LIN {X 0,Y 520.431,Z 549.53,A -85,B 0,C 180,E1 4700.342,E2 4700.342} C_VEL
LIN {X 0,Y 520.238,Z 549.53,A -85,B 0,C 180,E1 4705.945,E2 4705.945} C_VEL
LIN {X 0,Y 520.316,Z 549.53,A -85,B 0,C 180,E1 4711.444,E2 4711.444} C_VEL
LIN {X 0,Y 520.292,Z 549.53,A -85,B 0,C 180,E1 4717.494,E2 4717.494} C_VEL
LIN {X 0,Y 520.138,Z 549.53,A -85,B 0,C 180,E1 4723.505,E2 4723.505} C_VEL
LIN {X 0,Y 520.209,Z 549.53,A -85,B 0,C 180,E1 4728.919,E2 4728.919} C_VEL
LIN {X 0,Y 520.347,Z 549.53,A -85,B 0,C 180,E1 4734.548,E2 4734.548} C_VEL
LIN {X 0,Y 520.315,Z 549.53,A -85,B 0,C 180,E1 4740.458,E2 4740.458} C_VEL
LIN {X 0,Y 520.326,Z 549.53,A -85,B 0,C 180,E1 4746.044,E2 4746.044} C_VEL
LIN {X 0,Y 520.448,Z 549.53,A -85,B 0,C 180,E1 4751.4,E2 4751.4} C_VEL
LIN {X 0,Y 520.57,Z 549.53,A -85,B 0,C 180,E1 4756.59,E2 4756.59} C_VEL
LIN {X 0,Y 520.643,Z 549.53,A -85,B 0,C 180,E1 4761.666,E2 4761.666} C_VEL
LIN {X 0,Y 520.778,Z 549.53,A -85,B 0,C 180,E1 4766.365,E2 4766.365} C_VEL
LIN {X 0,Y 530.305,Z 577.59,A -85,B 0,C 180,E1 4767.616,E2 4767.616} C_VEL
LIN {X 0,Y 528.887,Z 613.589,A -85,B 0,C 180,E1 4768.906,E2 4768.906} C_VEL
LIN {X 0,Y 527.091,Z 649.664,A -85,B 0,C 180,E1 4770.921,E2 4770.921} C_VEL
LIN {X 0,Y 525.182,Z 681.953,A -85,B 0,C 180,E1 4773.499,E2 4773.499} C_VEL
LIN {X 0,Y 523.571,Z 709.362,A -85,B 0,C 180,E1 4776.451,E2 4776.451} C_VEL
LIN {X 0,Y 522.327,Z 733.847,A -85,B 0,C 180,E1 4779.981,E2 4779.981} C_VEL
LIN {X 0,Y 521.528,Z 752.418,A -85,B 0,C 180,E1 4783.667,E2 4783.667} C_VEL
LIN {X 0,Y 521.153,Z 765.124,A -85,B 0,C 180,E1 4787.243,E2 4787.243} C_VEL
LIN {X 0,Y 520.901,Z 773.821,A -85,B 0,C 180,E1 4791.198,E2 4791.198} C_VEL
LIN {X 0,Y 520.663,Z 776.795,A -85,B 0,C 180,E1 4793.937,E2 4793.937} C_VEL
LIN {X 0,Y 520.691,Z 777.009,A -85,B 0,C 180,E1 4797.624,E2 4797.624} C_VEL
LIN {X 0,Y 520.92,Z 772.639,A -85,B 0,C 180,E1 4801.427,E2 4801.427} C_VEL
LIN {X 0,Y 521.187,Z 762.933,A -85,B 0,C 180,E1 4805.383,E2 4805.383} C_VEL
LIN {X 0,Y 521.63,Z 747.74,A -85,B 0,C 180,E1 4809.291,E2 4809.291} C_VEL
LIN {X 0,Y 522.565,Z 727.336,A -85,B 0,C 180,E1 4812.983,E2 4812.983} C_VEL
LIN {X 0,Y 524.021,Z 701.188,A -85,B 0,C 180,E1 4816.431,E2 4816.431} C_VEL
LIN {X 0,Y 525.82,Z 671.672,A -85,B 0,C 180,E1 4819.322,E2 4819.322} C_VEL
LIN {X 0,Y 527.771,Z 637.844,A -85,B 0,C 180,E1 4821.735,E2 4821.735} C_VEL
LIN {X 0,Y 529.434,Z 602.923,A -85,B 0,C 180,E1 4823.452,E2 4823.452} C_VEL
LIN {X 0,Y 529.834,Z 574.051,A -85,B 0,C 180,E1 4824.43,E2 4824.43} C_VEL
LIN {X 0,Y 520.283,Z 549.53,A -85,B 0,C 180,E1 4825.673,E2 4825.673} C_VEL
LIN {X 0,Y 520.236,Z 549.53,A -85,B 0,C 180,E1 4832.371,E2 4832.371} C_VEL
LIN {X 0,Y 520.407,Z 549.53,A -85,B 0,C 180,E1 4838.106,E2 4838.106} C_VEL
LIN {X 0,Y 520.506,Z 549.53,A -85,B 0,C 180,E1 4843.166,E2 4843.166} C_VEL
LIN {X 0,Y 520.57,Z 549.53,A -85,B 0,C 180,E1 4850.251,E2 4850.251} C_VEL
LIN {X 0,Y 520.727,Z 549.53,A -85,B 0,C 180,E1 4855.028,E2 4855.028} C_VEL
LIN {X 0,Y 520.755,Z 549.53,A -85,B 0,C 180,E1 4860.014,E2 4860.014} C_VEL
LIN {X 0,Y 520.699,Z 549.53,A -85,B 0,C 180,E1 4865,E2 4865} C_VEL
LIN {X 0,Y 520.637,Z 549.53,A -85,B 0,C 180,E1 4870.027,E2 4870.027} C_VEL
LIN {X 0,Y 520.555,Z 549.53,A -85,B 0,C 180,E1 4875.134,E2 4875.134} C_VEL
LIN {X 0,Y 520.44,Z 549.53,A -85,B 0,C 180,E1 4880.371,E2 4880.371} C_VEL
LIN {X 0,Y 520.257,Z 549.53,A -85,B 0,C 180,E1 4885.955,E2 4885.955} C_VEL
LIN {X 0,Y 520.324,Z 549.53,A -85,B 0,C 180,E1 4891.476,E2 4891.476} C_VEL
LIN {X 0,Y 520.303,Z 549.53,A -85,B 0,C 180,E1 4894.283,E2 4894.283} C_VEL
LIN {X 0,Y 519.013,Z 549.53,A -85,B 0,C 180,E1 4895.236,E2 4895.236} C_VEL
LIN {X 0,Y 512.425,Z 549.53,A -85,B 0,C 180,E1 4897.832,E2 4897.832} C_VEL
LIN {X 0,Y 512.336,Z 549.53,A -85,B 0,C 180,E1 4898.078,E2 4898.078} C_VEL
LIN {X 0,Y 512.178,Z 549.53,A -85,B 0,C 180,E1 4902.666,E2 4902.666} C_VEL
LIN {X 0,Y 512.279,Z 549.53,A -85,B 0,C 180,E1 4909.607,E2 4909.607} C_VEL
LIN {X 0,Y 512.456,Z 549.825,A -85,B 0,C 180,E1 4914.218,E2 4914.218} C_VEL
LIN {X 0,Y 527.474,Z 581.593,A -85,B 0,C 180,E1 4915.838,E2 4915.838} C_VEL
LIN {X 0,Y 526.712,Z 627.123,A -85,B 0,C 180,E1 4916.726,E2 4916.726} C_VEL
LIN {X 0,Y 525.021,Z 664.478,A -85,B 0,C 180,E1 4918.051,E2 4918.051} C_VEL
LIN {X 0,Y 522.723,Z 701.045,A -85,B 0,C 180,E1 4920.007,E2 4920.007} C_VEL
LIN {X 0,Y 520.135,Z 735.661,A -85,B 0,C 180,E1 4922.578,E2 4922.578} C_VEL
LIN {X 0,Y 517.704,Z 767.36,A -85,B 0,C 180,E1 4925.726,E2 4925.726} C_VEL
LIN {X 0,Y 515.731,Z 794.257,A -85,B 0,C 180,E1 4929.222,E2 4929.222} C_VEL
LIN {X 0,Y 514.27,Z 817.275,A -85,B 0,C 180,E1 4933.158,E2 4933.158} C_VEL
LIN {X 0,Y 513.463,Z 834.988,A -85,B 0,C 180,E1 4937.268,E2 4937.268} C_VEL
LIN {X 0,Y 513.159,Z 847.681,A -85,B 0,C 180,E1 4941.546,E2 4941.546} C_VEL
LIN {X 0,Y 512.986,Z 853.959,A -85,B 0,C 180,E1 4944.938,E2 4944.938} C_VEL
LIN {X 0,Y 513.008,Z 857.089,A -85,B 0,C 180,E1 4948.316,E2 4948.316} C_VEL
LIN {X 0,Y 513.123,Z 857.088,A -85,B 0,C 180,E1 4951.686,E2 4951.686} C_VEL
LIN {X 0,Y 513.106,Z 852.753,A -85,B 0,C 180,E1 4955.909,E2 4955.909} C_VEL
LIN {X 0,Y 513.227,Z 843.301,A -85,B 0,C 180,E1 4960.162,E2 4960.162} C_VEL
LIN {X 0,Y 513.73,Z 829.231,A -85,B 0,C 180,E1 4964.223,E2 4964.223} C_VEL
LIN {X 0,Y 514.776,Z 809.386,A -85,B 0,C 180,E1 4968.323,E2 4968.323} C_VEL
LIN {X 0,Y 516.501,Z 783.307,A -85,B 0,C 180,E1 4972.323,E2 4972.323} C_VEL
LIN {X 0,Y 518.848,Z 752.442,A -85,B 0,C 180,E1 4975.867,E2 4975.867} C_VEL
LIN {X 0,Y 521.372,Z 718.916,A -85,B 0,C 180,E1 4978.764,E2 4978.764} C_VEL
LIN {X 0,Y 523.845,Z 683.514,A -85,B 0,C 180,E1 4981.019,E2 4981.019} C_VEL
LIN {X 0,Y 525.934,Z 646.139,A -85,B 0,C 180,E1 4982.677,E2 4982.677} C_VEL
LIN {X 0,Y 527.415,Z 608.302,A -85,B 0,C 180,E1 4983.705,E2 4983.705} C_VEL
LIN {X 0,Y 526.934,Z 580.932,A -85,B 0,C 180,E1 4984.213,E2 4984.213} C_VEL
LIN {X 0,Y 512.332,Z 549.53,A -85,B 0,C 180,E1 4985.885,E2 4985.885} C_VEL
LIN {X 0,Y 512.274,Z 549.53,A -85,B 0,C 180,E1 4990.397,E2 4990.397} C_VEL
LIN {X 0,Y 512.235,Z 549.53,A -85,B 0,C 180,E1 4995,E2 4995} C_VEL
LIN {X 0,Y 512.309,Z 549.53,A -85,B 0,C 180,E1 4999.983,E2 4999.983} C_VEL
LIN {X 0,Y 512.197,Z 549.53,A -85,B 0,C 180,E1 5005.952,E2 5005.952} C_VEL
LIN {X 0,Y 512.321,Z 549.53,A -85,B 0,C 180,E1 5012.086,E2 5012.086} C_VEL
LIN {X 0,Y 512.392,Z 549.53,A -85,B 0,C 180,E1 5017.48,E2 5017.48} C_VEL
LIN {X 0,Y 512.603,Z 549.53,A -85,B 0,C 180,E1 5022.869,E2 5022.869} C_VEL
LIN {X 0,Y 512.625,Z 549.53,A -85,B 0,C 180,E1 5029.815,E2 5029.815} C_VEL
LIN {X 0,Y 512.82,Z 549.53,A -85,B 0,C 180,E1 5034.923,E2 5034.923} C_VEL
LIN {X 0,Y 512.87,Z 549.53,A -85,B 0,C 180,E1 5039.986,E2 5039.986} C_VEL
LIN {X 0,Y 512.809,Z 549.53,A -85,B 0,C 180,E1 5045.049,E2 5045.049} C_VEL
LIN {X 0,Y 512.695,Z 549.53,A -85,B 0,C 180,E1 5050.155,E2 5050.155} C_VEL
LIN {X 0,Y 512.614,Z 549.53,A -85,B 0,C 180,E1 5055.345,E2 5055.345} C_VEL
LIN {X 0,Y 512.524,Z 549.53,A -85,B 0,C 180,E1 5060.67,E2 5060.67} C_VEL
LIN {X 0,Y 512.323,Z 549.53,A -85,B 0,C 180,E1 5066.197,E2 5066.197} C_VEL
LIN {X 0,Y 512.439,Z 549.53,A -85,B 0,C 180,E1 5071.984,E2 5071.984} C_VEL
LIN {X 0,Y 512.352,Z 549.53,A -85,B 0,C 180,E1 5078.179,E2 5078.179} C_VEL
LIN {X 0,Y 512.22,Z 549.53,A -85,B 0,C 180,E1 5082.624,E2 5082.624} C_VEL
LIN {X 0,Y 512.305,Z 549.53,A -85,B 0,C 180,E1 5089.606,E2 5089.606} C_VEL
LIN {X 0,Y 512.429,Z 549.53,A -85,B 0,C 180,E1 5095.976,E2 5095.976} C_VEL
LIN {X 0,Y 512.337,Z 549.53,A -85,B 0,C 180,E1 5102.025,E2 5102.025} C_VEL
LIN {X 0,Y 512.409,Z 549.53,A -85,B 0,C 180,E1 5107.489,E2 5107.489} C_VEL
LIN {X 0,Y 512.544,Z 549.53,A -85,B 0,C 180,E1 5112.876,E2 5112.876} C_VEL
LIN {X 0,Y 512.601,Z 549.53,A -85,B 0,C 180,E1 5118.107,E2 5118.107} C_VEL
LIN {X 0,Y 512.672,Z 549.53,A -85,B 0,C 180,E1 5123.237,E2 5123.237} C_VEL
LIN {X 0,Y 512.818,Z 549.53,A -85,B 0,C 180,E1 5125.81,E2 5125.81} C_VEL
LIN {X 0,Y 523.408,Z 579.421,A -85,B 0,C 180,E1 5127.229,E2 5127.229} C_VEL
LIN {X 0,Y 521.746,Z 616.27,A -85,B 0,C 180,E1 5128.616,E2 5128.616} C_VEL
LIN {X 0,Y 519.675,Z 652.179,A -85,B 0,C 180,E1 5130.727,E2 5130.727} C_VEL
LIN {X 0,Y 517.64,Z 683.856,A -85,B 0,C 180,E1 5133.341,E2 5133.341} C_VEL
LIN {X 0,Y 515.857,Z 712.071,A -85,B 0,C 180,E1 5136.492,E2 5136.492} C_VEL
LIN {X 0,Y 514.468,Z 736.085,A -85,B 0,C 180,E1 5140.135,E2 5140.135} C_VEL
LIN {X 0,Y 513.598,Z 754.208,A -85,B 0,C 180,E1 5143.919,E2 5143.919} C_VEL
LIN {X 0,Y 513.178,Z 767.479,A -85,B 0,C 180,E1 5147.983,E2 5147.983} C_VEL
LIN {X 0,Y 512.95,Z 774.361,A -85,B 0,C 180,E1 5151.504,E2 5151.504} C_VEL
LIN {X 0,Y 512.721,Z 777.052,A -85,B 0,C 180,E1 5154.332,E2 5154.332} C_VEL
LIN {X 0,Y 512.769,Z 776.742,A -85,B 0,C 180,E1 5158.089,E2 5158.089} C_VEL
LIN {X 0,Y 513.041,Z 771.802,A -85,B 0,C 180,E1 5161.966,E2 5161.966} C_VEL
LIN {X 0,Y 513.312,Z 761.433,A -85,B 0,C 180,E1 5166.01,E2 5166.01} C_VEL
LIN {X 0,Y 513.915,Z 745.321,A -85,B 0,C 180,E1 5170.016,E2 5170.016} C_VEL
LIN {X 0,Y 515.009,Z 724.121,A -85,B 0,C 180,E1 5173.73,E2 5173.73} C_VEL
LIN {X 0,Y 516.685,Z 697.579,A -85,B 0,C 180,E1 5177.157,E2 5177.157} C_VEL
LIN {X 0,Y 518.761,Z 666.697,A -85,B 0,C 180,E1 5180.088,E2 5180.088} C_VEL
LIN {X 0,Y 520.898,Z 633.126,A -85,B 0,C 180,E1 5182.396,E2 5182.396} C_VEL
LIN {X 0,Y 522.706,Z 598.792,A -85,B 0,C 180,E1 5184.046,E2 5184.046} C_VEL
LIN {X 0,Y 522.91,Z 576.09,A -85,B 0,C 180,E1 5184.826,E2 5184.826} C_VEL
LIN {X 0,Y 512.328,Z 549.53,A -85,B 0,C 180,E1 5186.174,E2 5186.174} C_VEL
LIN {X 0,Y 512.295,Z 549.53,A -85,B 0,C 180,E1 5192.086,E2 5192.086} C_VEL
LIN {X 0,Y 512.417,Z 549.53,A -85,B 0,C 180,E1 5197.511,E2 5197.511} C_VEL
LIN {X 0,Y 512.607,Z 549.53,A -85,B 0,C 180,E1 5202.898,E2 5202.898} C_VEL
LIN {X 0,Y 512.606,Z 549.53,A -85,B 0,C 180,E1 5209.843,E2 5209.843} C_VEL
LIN {X 0,Y 512.836,Z 549.53,A -85,B 0,C 180,E1 5214.951,E2 5214.951} C_VEL
LIN {X 0,Y 512.884,Z 549.53,A -85,B 0,C 180,E1 5220.014,E2 5220.014} C_VEL
LIN {X 0,Y 512.81,Z 549.53,A -85,B 0,C 180,E1 5225.077,E2 5225.077} C_VEL
LIN {X 0,Y 512.711,Z 549.53,A -85,B 0,C 180,E1 5230.183,E2 5230.183} C_VEL
LIN {X 0,Y 512.619,Z 549.53,A -85,B 0,C 180,E1 5235.374,E2 5235.374} C_VEL
LIN {X 0,Y 512.541,Z 549.53,A -85,B 0,C 180,E1 5240.699,E2 5240.699} C_VEL
LIN {X 0,Y 512.342,Z 549.53,A -85,B 0,C 180,E1 5246.228,E2 5246.228} C_VEL
LIN {X 0,Y 512.458,Z 549.53,A -85,B 0,C 180,E1 5252.016,E2 5252.016} C_VEL
LIN {X 0,Y 512.336,Z 549.53,A -85,B 0,C 180,E1 5258.078,E2 5258.078} C_VEL
LIN {X 0,Y 509.798,Z 549.53,A -85,B 0,C 180,E1 5259.506,E2 5259.506} C_VEL
LIN {X 0,Y 504.179,Z 549.53,A -85,B 0,C 180,E1 5261.893,E2 5261.893} C_VEL
LIN {X 0,Y 504.248,Z 549.53,A -85,B 0,C 180,E1 5268.437,E2 5268.437} C_VEL
LIN {X 0,Y 504.52,Z 550.06,A -85,B 0,C 180,E1 5273.641,E2 5273.641} C_VEL
LIN {X 0,Y 520.972,Z 585.329,A -85,B 0,C 180,E1 5275.412,E2 5275.412} C_VEL
LIN {X 0,Y 520.005,Z 629.452,A -85,B 0,C 180,E1 5276.313,E2 5276.313} C_VEL
LIN {X 0,Y 518.202,Z 665.289,A -85,B 0,C 180,E1 5277.621,E2 5277.621} C_VEL
LIN {X 0,Y 515.74,Z 701.042,A -85,B 0,C 180,E1 5279.558,E2 5279.558} C_VEL
LIN {X 0,Y 512.874,Z 736.63,A -85,B 0,C 180,E1 5282.248,E2 5282.248} C_VEL
LIN {X 0,Y 510.284,Z 767.554,A -85,B 0,C 180,E1 5285.374,E2 5285.374} C_VEL
LIN {X 0,Y 508.141,Z 794.257,A -85,B 0,C 180,E1 5288.897,E2 5288.897} C_VEL
LIN {X 0,Y 506.557,Z 817.274,A -85,B 0,C 180,E1 5292.893,E2 5292.893} C_VEL
LIN {X 0,Y 505.642,Z 834.989,A -85,B 0,C 180,E1 5297.067,E2 5297.067} C_VEL
LIN {X 0,Y 505.268,Z 847.681,A -85,B 0,C 180,E1 5301.413,E2 5301.413} C_VEL
LIN {X 0,Y 505.092,Z 853.959,A -85,B 0,C 180,E1 5304.859,E2 5304.859} C_VEL
LIN {X 0,Y 505.105,Z 857.089,A -85,B 0,C 180,E1 5308.289,E2 5308.289} C_VEL
LIN {X 0,Y 505.216,Z 857.088,A -85,B 0,C 180,E1 5311.713,E2 5311.713} C_VEL
LIN {X 0,Y 505.215,Z 852.753,A -85,B 0,C 180,E1 5316.002,E2 5316.002} C_VEL
LIN {X 0,Y 505.34,Z 843.301,A -85,B 0,C 180,E1 5320.323,E2 5320.323} C_VEL
LIN {X 0,Y 505.98,Z 828.122,A -85,B 0,C 180,E1 5324.727,E2 5324.727} C_VEL
LIN {X 0,Y 507.267,Z 806.651,A -85,B 0,C 180,E1 5329.102,E2 5329.102} C_VEL
LIN {X 0,Y 509.104,Z 781.479,A -85,B 0,C 180,E1 5332.911,E2 5332.911} C_VEL
LIN {X 0,Y 511.641,Z 751.299,A -85,B 0,C 180,E1 5336.377,E2 5336.377} C_VEL
LIN {X 0,Y 514.409,Z 717.39,A -85,B 0,C 180,E1 5339.31,E2 5339.31} C_VEL
LIN {X 0,Y 517.157,Z 681.161,A -85,B 0,C 180,E1 5341.601,E2 5341.601} C_VEL
LIN {X 0,Y 519.355,Z 643.386,A -85,B 0,C 180,E1 5343.249,E2 5343.249} C_VEL
LIN {X 0,Y 520.93,Z 604.752,A -85,B 0,C 180,E1 5344.251,E2 5344.251} C_VEL
LIN {X 0,Y 520.343,Z 583.478,A -85,B 0,C 180,E1 5344.666,E2 5344.666} C_VEL
LIN {X 0,Y 504.411,Z 549.53,A -85,B 0,C 180,E1 5346.469,E2 5346.469} C_VEL
LIN {X 0,Y 504.253,Z 549.53,A -85,B 0,C 180,E1 5351.564,E2 5351.564} C_VEL
LIN {X 0,Y 504.254,Z 549.53,A -85,B 0,C 180,E1 5356.498,E2 5356.498} C_VEL
LIN {X 0,Y 504.376,Z 549.53,A -85,B 0,C 180,E1 5361.069,E2 5361.069} C_VEL
LIN {X 0,Y 504.26,Z 549.53,A -85,B 0,C 180,E1 5366.922,E2 5366.922} C_VEL
LIN {X 0,Y 504.383,Z 549.53,A -85,B 0,C 180,E1 5373.326,E2 5373.326} C_VEL
LIN {X 0,Y 504.551,Z 549.53,A -85,B 0,C 180,E1 5378.957,E2 5378.957} C_VEL
LIN {X 0,Y 504.545,Z 549.53,A -85,B 0,C 180,E1 5384.374,E2 5384.374} C_VEL
LIN {X 0,Y 504.688,Z 549.53,A -85,B 0,C 180,E1 5390.652,E2 5390.652} C_VEL
LIN {X 0,Y 504.879,Z 549.53,A -85,B 0,C 180,E1 5396.56,E2 5396.56} C_VEL
LIN {X 0,Y 504.89,Z 549.53,A -85,B 0,C 180,E1 5401.698,E2 5401.698} C_VEL
LIN {X 0,Y 504.798,Z 549.53,A -85,B 0,C 180,E1 5406.852,E2 5406.852} C_VEL
LIN {X 0,Y 504.725,Z 549.53,A -85,B 0,C 180,E1 5412.063,E2 5412.063} C_VEL
LIN {X 0,Y 504.672,Z 549.53,A -85,B 0,C 180,E1 5417.379,E2 5417.379} C_VEL
LIN {X 0,Y 504.522,Z 549.53,A -85,B 0,C 180,E1 5422.86,E2 5422.86} C_VEL
LIN {X 0,Y 504.409,Z 549.53,A -85,B 0,C 180,E1 5428.575,E2 5428.575} C_VEL
LIN {X 0,Y 504.512,Z 549.53,A -85,B 0,C 180,E1 5434.605,E2 5434.605} C_VEL
LIN {X 0,Y 504.301,Z 549.53,A -85,B 0,C 180,E1 5441.14,E2 5441.14} C_VEL
LIN {X 0,Y 504.2,Z 549.53,A -85,B 0,C 180,E1 5446.498,E2 5446.498} C_VEL
LIN {X 0,Y 504.461,Z 549.53,A -85,B 0,C 180,E1 5453.252,E2 5453.252} C_VEL
LIN {X 0,Y 504.481,Z 549.53,A -85,B 0,C 180,E1 5459.434,E2 5459.434} C_VEL
LIN {X 0,Y 504.416,Z 549.53,A -85,B 0,C 180,E1 5465.238,E2 5465.238} C_VEL
LIN {X 0,Y 504.573,Z 549.53,A -85,B 0,C 180,E1 5470.792,E2 5470.792} C_VEL
LIN {X 0,Y 504.731,Z 549.53,A -85,B 0,C 180,E1 5476.161,E2 5476.161} C_VEL
LIN {X 0,Y 504.802,Z 549.53,A -85,B 0,C 180,E1 5481.403,E2 5481.403} C_VEL
LIN {X 0,Y 504.918,Z 549.53,A -85,B 0,C 180,E1 5485.252,E2 5485.252} C_VEL
LIN {X 0,Y 516.561,Z 581.031,A -85,B 0,C 180,E1 5486.825,E2 5486.825} C_VEL
LIN {X 0,Y 514.777,Z 617.903,A -85,B 0,C 180,E1 5488.251,E2 5488.251} C_VEL
LIN {X 0,Y 512.468,Z 653.021,A -85,B 0,C 180,E1 5490.378,E2 5490.378} C_VEL
LIN {X 0,Y 509.988,Z 686.88,A -85,B 0,C 180,E1 5493.285,E2 5493.285} C_VEL
LIN {X 0,Y 508.003,Z 715.033,A -85,B 0,C 180,E1 5496.593,E2 5496.593} C_VEL
LIN {X 0,Y 506.654,Z 737.121,A -85,B 0,C 180,E1 5500.076,E2 5500.076} C_VEL
LIN {X 0,Y 505.694,Z 755.846,A -85,B 0,C 180,E1 5504.141,E2 5504.141} C_VEL
LIN {X 0,Y 505.266,Z 768.495,A -85,B 0,C 180,E1 5508.274,E2 5508.274} C_VEL
LIN {X 0,Y 504.949,Z 775.337,A -85,B 0,C 180,E1 5512.188,E2 5512.188} C_VEL
LIN {X 0,Y 504.819,Z 777.436,A -85,B 0,C 180,E1 5516.324,E2 5516.324} C_VEL
LIN {X 0,Y 505.082,Z 774.295,A -85,B 0,C 180,E1 5520.523,E2 5520.523} C_VEL
LIN {X 0,Y 505.401,Z 766.132,A -85,B 0,C 180,E1 5524.56,E2 5524.56} C_VEL
LIN {X 0,Y 505.874,Z 751.801,A -85,B 0,C 180,E1 5528.785,E2 5528.785} C_VEL
LIN {X 0,Y 506.827,Z 732.332,A -85,B 0,C 180,E1 5532.687,E2 5532.687} C_VEL
LIN {X 0,Y 508.508,Z 707.772,A -85,B 0,C 180,E1 5536.267,E2 5536.267} C_VEL
LIN {X 0,Y 510.638,Z 677.998,A -85,B 0,C 180,E1 5539.478,E2 5539.478} C_VEL
LIN {X 0,Y 513.09,Z 645.394,A -85,B 0,C 180,E1 5542.069,E2 5542.069} C_VEL
LIN {X 0,Y 515.188,Z 612.098,A -85,B 0,C 180,E1 5543.94,E2 5543.94} C_VEL
LIN {X 0,Y 516.197,Z 578.793,A -85,B 0,C 180,E1 5545.2,E2 5545.2} C_VEL
LIN {X 0,Y 504.391,Z 549.53,A -85,B 0,C 180,E1 5546.785,E2 5546.785} C_VEL
LIN {X 0,Y 504.375,Z 549.53,A -85,B 0,C 180,E1 5553.357,E2 5553.357} C_VEL
LIN {X 0,Y 504.589,Z 549.53,A -85,B 0,C 180,E1 5558.99,E2 5558.99} C_VEL
LIN {X 0,Y 504.533,Z 549.53,A -85,B 0,C 180,E1 5564.403,E2 5564.403} C_VEL
LIN {X 0,Y 504.678,Z 549.53,A -85,B 0,C 180,E1 5570.643,E2 5570.643} C_VEL
LIN {X 0,Y 504.861,Z 549.53,A -85,B 0,C 180,E1 5576.588,E2 5576.588} C_VEL
LIN {X 0,Y 504.834,Z 549.53,A -85,B 0,C 180,E1 5581.727,E2 5581.727} C_VEL
LIN {X 0,Y 504.805,Z 549.53,A -85,B 0,C 180,E1 5586.88,E2 5586.88} C_VEL
LIN {X 0,Y 504.739,Z 549.53,A -85,B 0,C 180,E1 5592.092,E2 5592.092} C_VEL
LIN {X 0,Y 504.669,Z 549.53,A -85,B 0,C 180,E1 5597.409,E2 5597.409} C_VEL
LIN {X 0,Y 504.513,Z 549.53,A -85,B 0,C 180,E1 5602.892,E2 5602.892} C_VEL
LIN {X 0,Y 504.415,Z 549.53,A -85,B 0,C 180,E1 5608.607,E2 5608.607} C_VEL
LIN {X 0,Y 504.495,Z 549.53,A -85,B 0,C 180,E1 5614.641,E2 5614.641} C_VEL
LIN {X 0,Y 504.249,Z 549.53,A -85,B 0,C 180,E1 5621.183,E2 5621.183} C_VEL
LIN {X 0,Y 504.179,Z 549.53,A -85,B 0,C 180,E1 5621.893,E2 5621.893} C_VEL
LIN {X 0,Y 500.185,Z 549.53,A -85,B 0,C 180,E1 5623.841,E2 5623.841} C_VEL
LIN {X 0,Y 496.251,Z 549.53,A -85,B 0,C 180,E1 5625.819,E2 5625.819} C_VEL
LIN {X 0,Y 496.471,Z 549.53,A -85,B 0,C 180,E1 5632.216,E2 5632.216} C_VEL
LIN {X 0,Y 496.589,Z 550.219,A -85,B 0,C 180,E1 5633.041,E2 5633.041} C_VEL
LIN {X 0,Y 514.376,Z 587.202,A -85,B 0,C 180,E1 5634.958,E2 5634.958} C_VEL
LIN {X 0,Y 513.394,Z 630.256,A -85,B 0,C 180,E1 5635.846,E2 5635.846} C_VEL
LIN {X 0,Y 511.362,Z 666.981,A -85,B 0,C 180,E1 5637.222,E2 5637.222} C_VEL
LIN {X 0,Y 508.583,Z 704.006,A -85,B 0,C 180,E1 5639.299,E2 5639.299} C_VEL
LIN {X 0,Y 505.529,Z 738.494,A -85,B 0,C 180,E1 5641.989,E2 5641.989} C_VEL
LIN {X 0,Y 502.776,Z 768.957,A -85,B 0,C 180,E1 5645.155,E2 5645.155} C_VEL
LIN {X 0,Y 500.443,Z 795.709,A -85,B 0,C 180,E1 5648.788,E2 5648.788} C_VEL
LIN {X 0,Y 498.731,Z 818.354,A -85,B 0,C 180,E1 5652.843,E2 5652.843} C_VEL
LIN {X 0,Y 497.81,Z 834.989,A -85,B 0,C 180,E1 5656.86,E2 5656.86} C_VEL
LIN {X 0,Y 497.394,Z 847.681,A -85,B 0,C 180,E1 5661.276,E2 5661.276} C_VEL
LIN {X 0,Y 497.2,Z 853.959,A -85,B 0,C 180,E1 5664.777,E2 5664.777} C_VEL
LIN {X 0,Y 497.229,Z 857.089,A -85,B 0,C 180,E1 5668.262,E2 5668.262} C_VEL
LIN {X 0,Y 497.313,Z 857.088,A -85,B 0,C 180,E1 5671.74,E2 5671.74} C_VEL
LIN {X 0,Y 497.338,Z 852.753,A -85,B 0,C 180,E1 5676.097,E2 5676.097} C_VEL
LIN {X 0,Y 497.452,Z 843.301,A -85,B 0,C 180,E1 5680.488,E2 5680.488} C_VEL
LIN {X 0,Y 498.224,Z 827.671,A -85,B 0,C 180,E1 5685.077,E2 5685.077} C_VEL
LIN {X 0,Y 499.615,Z 806.649,A -85,B 0,C 180,E1 5689.406,E2 5689.406} C_VEL
LIN {X 0,Y 501.63,Z 781.478,A -85,B 0,C 180,E1 5693.272,E2 5693.272} C_VEL
LIN {X 0,Y 504.348,Z 751.407,A -85,B 0,C 180,E1 5696.777,E2 5696.777} C_VEL
LIN {X 0,Y 507.259,Z 718.909,A -85,B 0,C 180,E1 5699.643,E2 5699.643} C_VEL
LIN {X 0,Y 510.196,Z 683.124,A -85,B 0,C 180,E1 5701.968,E2 5701.968} C_VEL
LIN {X 0,Y 512.617,Z 645.726,A -85,B 0,C 180,E1 5703.653,E2 5703.653} C_VEL
LIN {X 0,Y 514.296,Z 608.516,A -85,B 0,C 180,E1 5704.673,E2 5704.673} C_VEL
LIN {X 0,Y 514.031,Z 586.652,A -85,B 0,C 180,E1 5705.079,E2 5705.079} C_VEL
LIN {X 0,Y 496.607,Z 551.017,A -85,B 0,C 180,E1 5706.98,E2 5706.98} C_VEL
LIN {X 0,Y 496.464,Z 549.53,A -85,B 0,C 180,E1 5707.02,E2 5707.02} C_VEL
LIN {X 0,Y 496.307,Z 549.53,A -85,B 0,C 180,E1 5713.131,E2 5713.131} C_VEL
LIN {X 0,Y 496.351,Z 549.53,A -85,B 0,C 180,E1 5719.471,E2 5719.471} C_VEL
LIN {X 0,Y 496.401,Z 549.53,A -85,B 0,C 180,E1 5725.165,E2 5725.165} C_VEL
LIN {X 0,Y 496.412,Z 549.53,A -85,B 0,C 180,E1 5731.833,E2 5731.833} C_VEL
LIN {X 0,Y 496.504,Z 549.53,A -85,B 0,C 180,E1 5736.717,E2 5736.717} C_VEL
LIN {X 0,Y 496.756,Z 549.53,A -85,B 0,C 180,E1 5742.305,E2 5742.305} C_VEL
LIN {X 0,Y 496.772,Z 549.53,A -85,B 0,C 180,E1 5749.486,E2 5749.486} C_VEL
LIN {X 0,Y 497.015,Z 549.53,A -85,B 0,C 180,E1 5754.761,E2 5754.761} C_VEL
LIN {X 0,Y 497.077,Z 549.53,A -85,B 0,C 180,E1 5759.986,E2 5759.986} C_VEL
LIN {X 0,Y 496.994,Z 549.53,A -85,B 0,C 180,E1 5765.21,E2 5765.21} C_VEL
LIN {X 0,Y 496.858,Z 549.53,A -85,B 0,C 180,E1 5770.482,E2 5770.482} C_VEL
LIN {X 0,Y 496.768,Z 549.53,A -85,B 0,C 180,E1 5775.847,E2 5775.847} C_VEL
LIN {X 0,Y 496.641,Z 549.53,A -85,B 0,C 180,E1 5781.363,E2 5781.363} C_VEL
LIN {X 0,Y 496.454,Z 549.53,A -85,B 0,C 180,E1 5787.102,E2 5787.102} C_VEL
LIN {X 0,Y 496.554,Z 549.53,A -85,B 0,C 180,E1 5793.136,E2 5793.136} C_VEL
LIN {X 0,Y 496.405,Z 549.53,A -85,B 0,C 180,E1 5799.641,E2 5799.641} C_VEL
LIN {X 0,Y 496.303,Z 549.53,A -85,B 0,C 180,E1 5805.626,E2 5805.626} C_VEL
LIN {X 0,Y 496.462,Z 549.53,A -85,B 0,C 180,E1 5812.17,E2 5812.17} C_VEL
LIN {X 0,Y 496.554,Z 549.53,A -85,B 0,C 180,E1 5816.836,E2 5816.836} C_VEL
LIN {X 0,Y 496.44,Z 549.53,A -85,B 0,C 180,E1 5822.872,E2 5822.872} C_VEL
LIN {X 0,Y 496.585,Z 549.53,A -85,B 0,C 180,E1 5828.612,E2 5828.612} C_VEL
LIN {X 0,Y 496.748,Z 549.53,A -85,B 0,C 180,E1 5834.132,E2 5834.132} C_VEL
LIN {X 0,Y 496.815,Z 549.53,A -85,B 0,C 180,E1 5839.498,E2 5839.498} C_VEL
LIN {X 0,Y 496.95,Z 549.53,A -85,B 0,C 180,E1 5844.663,E2 5844.663} C_VEL
LIN {X 0,Y 509.701,Z 582.361,A -85,B 0,C 180,E1 5846.399,E2 5846.399} C_VEL
LIN {X 0,Y 507.802,Z 619.644,A -85,B 0,C 180,E1 5847.884,E2 5847.884} C_VEL
LIN {X 0,Y 505.351,Z 653.871,A -85,B 0,C 180,E1 5849.999,E2 5849.999} C_VEL
LIN {X 0,Y 502.82,Z 684.793,A -85,B 0,C 180,E1 5852.686,E2 5852.686} C_VEL
LIN {X 0,Y 500.522,Z 713.378,A -85,B 0,C 180,E1 5856.054,E2 5856.054} C_VEL
LIN {X 0,Y 498.939,Z 736.959,A -85,B 0,C 180,E1 5859.794,E2 5859.794} C_VEL
LIN {X 0,Y 497.919,Z 754.399,A -85,B 0,C 180,E1 5863.583,E2 5863.583} C_VEL
LIN {X 0,Y 497.428,Z 767.297,A -85,B 0,C 180,E1 5867.658,E2 5867.658} C_VEL
LIN {X 0,Y 497.121,Z 774.359,A -85,B 0,C 180,E1 5871.361,E2 5871.361} C_VEL
LIN {X 0,Y 496.868,Z 777.353,A -85,B 0,C 180,E1 5875.161,E2 5875.161} C_VEL
LIN {X 0,Y 497.019,Z 776.045,A -85,B 0,C 180,E1 5879.062,E2 5879.062} C_VEL
LIN {X 0,Y 497.361,Z 769.937,A -85,B 0,C 180,E1 5883.1,E2 5883.1} C_VEL
LIN {X 0,Y 497.772,Z 758.102,A -85,B 0,C 180,E1 5887.321,E2 5887.321} C_VEL
LIN {X 0,Y 498.679,Z 740.328,A -85,B 0,C 180,E1 5891.489,E2 5891.489} C_VEL
LIN {X 0,Y 500.171,Z 717.58,A -85,B 0,C 180,E1 5895.267,E2 5895.267} C_VEL
LIN {X 0,Y 502.584,Z 688.392,A -85,B 0,C 180,E1 5898.863,E2 5898.863} C_VEL
LIN {X 0,Y 505.111,Z 657.131,A -85,B 0,C 180,E1 5901.687,E2 5901.687} C_VEL
LIN {X 0,Y 507.627,Z 623.874,A -85,B 0,C 180,E1 5903.821,E2 5903.821} C_VEL
LIN {X 0,Y 509.671,Z 586.534,A -85,B 0,C 180,E1 5905.409,E2 5905.409} C_VEL
LIN {X 0,Y 508.673,Z 579.152,A -85,B 0,C 180,E1 5905.718,E2 5905.718} C_VEL
LIN {X 0,Y 496.446,Z 549.53,A -85,B 0,C 180,E1 5907.444,E2 5907.444} C_VEL
LIN {X 0,Y 496.41,Z 549.53,A -85,B 0,C 180,E1 5912.895,E2 5912.895} C_VEL
LIN {X 0,Y 496.647,Z 549.53,A -85,B 0,C 180,E1 5918.637,E2 5918.637} C_VEL
LIN {X 0,Y 496.649,Z 549.53,A -85,B 0,C 180,E1 5924.149,E2 5924.149} C_VEL
LIN {X 0,Y 496.751,Z 549.53,A -85,B 0,C 180,E1 5929.515,E2 5929.515} C_VEL
LIN {X 0,Y 497.025,Z 549.53,A -85,B 0,C 180,E1 5934.79,E2 5934.79} C_VEL
LIN {X 0,Y 497.081,Z 549.53,A -85,B 0,C 180,E1 5940.014,E2 5940.014} C_VEL
LIN {X 0,Y 496.996,Z 549.53,A -85,B 0,C 180,E1 5945.24,E2 5945.24} C_VEL
LIN {X 0,Y 496.875,Z 549.53,A -85,B 0,C 180,E1 5950.511,E2 5950.511} C_VEL
LIN {X 0,Y 496.766,Z 549.53,A -85,B 0,C 180,E1 5955.877,E2 5955.877} C_VEL
LIN {X 0,Y 496.662,Z 549.53,A -85,B 0,C 180,E1 5961.393,E2 5961.393} C_VEL
LIN {X 0,Y 496.478,Z 549.53,A -85,B 0,C 180,E1 5967.133,E2 5967.133} C_VEL
LIN {X 0,Y 496.564,Z 549.53,A -85,B 0,C 180,E1 5973.17,E2 5973.17} C_VEL
LIN {X 0,Y 496.336,Z 549.53,A -85,B 0,C 180,E1 5979.685,E2 5979.685} C_VEL
LIN {X 0,Y 496.251,Z 549.53,A -85,B 0,C 180,E1 5985.819,E2 5985.819} C_VEL
LIN {X 0,Y 492.324,Z 549.53,A -85,B 0,C 180,E1 5987.794,E2 5987.794} C_VEL
LIN {X 0,Y 488.427,Z 549.53,A -85,B 0,C 180,E1 5989.8,E2 5989.8} C_VEL
LIN {X 0,Y 488.577,Z 549.53,A -85,B 0,C 180,E1 5992.391,E2 5992.391} C_VEL
LIN {X 0,Y 499.836,Z 573.662,A -85,B 0,C 180,E1 5993.684,E2 5993.684} C_VEL
LIN {X 0,Y 507.693,Z 590.543,A -85,B 0,C 180,E1 5994.54,E2 5994.54} C_VEL
LIN {X 0,Y 506.516,Z 632.795,A -85,B 0,C 180,E1 5995.457,E2 5995.457} C_VEL
LIN {X 0,Y 504.331,Z 671.305,A -85,B 0,C 180,E1 5996.947,E2 5996.947} C_VEL
LIN {X 0,Y 501.477,Z 706.397,A -85,B 0,C 180,E1 5998.993,E2 5998.993} C_VEL
LIN {X 0,Y 498.198,Z 740.32,A -85,B 0,C 180,E1 6001.718,E2 6001.718} C_VEL
LIN {X 0,Y 495.224,Z 770.8,A -85,B 0,C 180,E1 6004.982,E2 6004.982} C_VEL
LIN {X 0,Y 492.583,Z 798.855,A -85,B 0,C 180,E1 6008.943,E2 6008.943} C_VEL
LIN {X 0,Y 490.801,Z 820.879,A -85,B 0,C 180,E1 6013.096,E2 6013.096} C_VEL
LIN {X 0,Y 489.802,Z 838.045,A -85,B 0,C 180,E1 6017.547,E2 6017.547} C_VEL
LIN {X 0,Y 489.457,Z 849.598,A -85,B 0,C 180,E1 6022.027,E2 6022.027} C_VEL
LIN {X 0,Y 489.302,Z 855.91,A -85,B 0,C 180,E1 6026.465,E2 6026.465} C_VEL
LIN {X 0,Y 489.329,Z 857.5,A -85,B 0,C 180,E1 6030.001,E2 6030.001} C_VEL
LIN {X 0,Y 489.295,Z 855.909,A -85,B 0,C 180,E1 6033.538,E2 6033.538} C_VEL
LIN {X 0,Y 489.477,Z 849.594,A -85,B 0,C 180,E1 6037.976,E2 6037.976} C_VEL
LIN {X 0,Y 489.902,Z 838.038,A -85,B 0,C 180,E1 6042.453,E2 6042.453} C_VEL
LIN {X 0,Y 490.905,Z 820.902,A -85,B 0,C 180,E1 6046.895,E2 6046.895} C_VEL
LIN {X 0,Y 492.641,Z 797.746,A -85,B 0,C 180,E1 6051.234,E2 6051.234} C_VEL
LIN {X 0,Y 495.208,Z 770.783,A -85,B 0,C 180,E1 6055.021,E2 6055.021} C_VEL
LIN {X 0,Y 498.199,Z 740.318,A -85,B 0,C 180,E1 6058.282,E2 6058.282} C_VEL
LIN {X 0,Y 501.315,Z 707.642,A -85,B 0,C 180,E1 6060.925,E2 6060.925} C_VEL
LIN {X 0,Y 504.234,Z 671.102,A -85,B 0,C 180,E1 6063.07,E2 6063.07} C_VEL
LIN {X 0,Y 506.452,Z 633.016,A -85,B 0,C 180,E1 6064.548,E2 6064.548} C_VEL
LIN {X 0,Y 507.647,Z 589.87,A -85,B 0,C 180,E1 6065.487,E2 6065.487} C_VEL
LIN {X 0,Y 488.523,Z 549.53,A -85,B 0,C 180,E1 6067.703,E2 6067.703} C_VEL
LIN {X 0,Y 488.397,Z 549.53,A -85,B 0,C 180,E1 6072.825,E2 6072.825} C_VEL
LIN {X 0,Y 488.436,Z 549.53,A -85,B 0,C 180,E1 6077.859,E2 6077.859} C_VEL
LIN {X 0,Y 488.416,Z 549.53,A -85,B 0,C 180,E1 6084.045,E2 6084.045} C_VEL
LIN {X 0,Y 488.431,Z 549.53,A -85,B 0,C 180,E1 6090.366,E2 6090.366} C_VEL
LIN {X 0,Y 488.583,Z 549.53,A -85,B 0,C 180,E1 6096.317,E2 6096.317} C_VEL
LIN {X 0,Y 488.814,Z 549.53,A -85,B 0,C 180,E1 6102.007,E2 6102.007} C_VEL
LIN {X 0,Y 488.722,Z 549.53,A -85,B 0,C 180,E1 6107.506,E2 6107.506} C_VEL
LIN {X 0,Y 489.064,Z 549.53,A -85,B 0,C 180,E1 6112.897,E2 6112.897} C_VEL
LIN {X 0,Y 489.329,Z 549.53,A -85,B 0,C 180,E1 6118.219,E2 6118.219} C_VEL
LIN {X 0,Y 489.199,Z 549.53,A -85,B 0,C 180,E1 6123.521,E2 6123.521} C_VEL
LIN {X 0,Y 488.969,Z 549.53,A -85,B 0,C 180,E1 6129.041,E2 6129.041} C_VEL
LIN {X 0,Y 488.936,Z 549.53,A -85,B 0,C 180,E1 6134.276,E2 6134.276} C_VEL
LIN {X 0,Y 488.758,Z 549.53,A -85,B 0,C 180,E1 6139.833,E2 6139.833} C_VEL
LIN {X 0,Y 488.556,Z 549.53,A -85,B 0,C 180,E1 6145.598,E2 6145.598} C_VEL
LIN {X 0,Y 488.598,Z 549.53,A -85,B 0,C 180,E1 6151.645,E2 6151.645} C_VEL
LIN {X 0,Y 488.535,Z 549.53,A -85,B 0,C 180,E1 6158.124,E2 6158.124} C_VEL
LIN {X 0,Y 488.41,Z 549.53,A -85,B 0,C 180,E1 6164.713,E2 6164.713} C_VEL
LIN {X 0,Y 488.486,Z 549.53,A -85,B 0,C 180,E1 6170.52,E2 6170.52} C_VEL
LIN {X 0,Y 488.629,Z 549.53,A -85,B 0,C 180,E1 6176.447,E2 6176.447} C_VEL
LIN {X 0,Y 488.526,Z 549.53,A -85,B 0,C 180,E1 6182.396,E2 6182.396} C_VEL
LIN {X 0,Y 488.633,Z 549.53,A -85,B 0,C 180,E1 6188.247,E2 6188.247} C_VEL
LIN {X 0,Y 488.805,Z 549.53,A -85,B 0,C 180,E1 6193.867,E2 6193.867} C_VEL
LIN {X 0,Y 488.902,Z 549.53,A -85,B 0,C 180,E1 6199.326,E2 6199.326} C_VEL
LIN {X 0,Y 489.009,Z 550.013,A -85,B 0,C 180,E1 6204.076,E2 6204.076} C_VEL
LIN {X 0,Y 502.655,Z 583.898,A -85,B 0,C 180,E1 6205.952,E2 6205.952} C_VEL
LIN {X 0,Y 500.816,Z 621.517,A -85,B 0,C 180,E1 6207.516,E2 6207.516} C_VEL
LIN {X 0,Y 498.285,Z 654.219,A -85,B 0,C 180,E1 6209.57,E2 6209.57} C_VEL
LIN {X 0,Y 495.572,Z 685.162,A -85,B 0,C 180,E1 6212.289,E2 6212.289} C_VEL
LIN {X 0,Y 493.091,Z 712.444,A -85,B 0,C 180,E1 6215.548,E2 6215.548} C_VEL
LIN {X 0,Y 491.159,Z 737.553,A -85,B 0,C 180,E1 6219.644,E2 6219.644} C_VEL
LIN {X 0,Y 489.998,Z 756.038,A -85,B 0,C 180,E1 6223.807,E2 6223.807} C_VEL
LIN {X 0,Y 489.536,Z 768.336,A -85,B 0,C 180,E1 6227.953,E2 6227.953} C_VEL
LIN {X 0,Y 489.106,Z 775.579,A -85,B 0,C 180,E1 6232.317,E2 6232.317} C_VEL
LIN {X 0,Y 488.905,Z 777.395,A -85,B 0,C 180,E1 6236.54,E2 6236.54} C_VEL
LIN {X 0,Y 489.25,Z 774.762,A -85,B 0,C 180,E1 6240.327,E2 6240.327} C_VEL
LIN {X 0,Y 489.613,Z 766.488,A -85,B 0,C 180,E1 6244.701,E2 6244.701} C_VEL
LIN {X 0,Y 490.162,Z 753.493,A -85,B 0,C 180,E1 6248.762,E2 6248.762} C_VEL
LIN {X 0,Y 491.222,Z 734.99,A -85,B 0,C 180,E1 6252.754,E2 6252.754} C_VEL
LIN {X 0,Y 493.279,Z 710.568,A -85,B 0,C 180,E1 6256.623,E2 6256.623} C_VEL
LIN {X 0,Y 495.74,Z 683.933,A -85,B 0,C 180,E1 6259.767,E2 6259.767} C_VEL
LIN {X 0,Y 498.449,Z 653.758,A -85,B 0,C 180,E1 6262.402,E2 6262.402} C_VEL
LIN {X 0,Y 501.207,Z 618.016,A -85,B 0,C 180,E1 6264.6,E2 6264.6} C_VEL
LIN {X 0,Y 502.564,Z 583.368,A -85,B 0,C 180,E1 6266.023,E2 6266.023} C_VEL
LIN {X 0,Y 488.488,Z 549.53,A -85,B 0,C 180,E1 6267.989,E2 6267.989} C_VEL
LIN {X 0,Y 488.525,Z 549.53,A -85,B 0,C 180,E1 6274.4,E2 6274.4} C_VEL
LIN {X 0,Y 488.799,Z 549.53,A -85,B 0,C 180,E1 6280.169,E2 6280.169} C_VEL
LIN {X 0,Y 488.661,Z 549.53,A -85,B 0,C 180,E1 6285.716,E2 6285.716} C_VEL
LIN {X 0,Y 488.909,Z 549.53,A -85,B 0,C 180,E1 6291.139,E2 6291.139} C_VEL
LIN {X 0,Y 489.07,Z 549.53,A -85,B 0,C 180,E1 6296.478,E2 6296.478} C_VEL
LIN {X 0,Y 489.057,Z 549.53,A -85,B 0,C 180,E1 6301.782,E2 6301.782} C_VEL
LIN {X 0,Y 489.006,Z 549.53,A -85,B 0,C 180,E1 6307.104,E2 6307.104} C_VEL
LIN {X 0,Y 488.944,Z 549.53,A -85,B 0,C 180,E1 6312.489,E2 6312.489} C_VEL
LIN {X 0,Y 488.79,Z 549.53,A -85,B 0,C 180,E1 6317.993,E2 6317.993} C_VEL
LIN {X 0,Y 488.652,Z 549.53,A -85,B 0,C 180,E1 6323.679,E2 6323.679} C_VEL
LIN {X 0,Y 488.534,Z 549.53,A -85,B 0,C 180,E1 6330.134,E2 6330.134} C_VEL
LIN {X 0,Y 488.567,Z 549.53,A -85,B 0,C 180,E1 6335.942,E2 6335.942} C_VEL
LIN {X 0,Y 488.377,Z 549.53,A -85,B 0,C 180,E1 6342.137,E2 6342.137} C_VEL
LIN {X 0,Y 488.392,Z 549.53,A -85,B 0,C 180,E1 6347.87,E2 6347.87} C_VEL
LIN {X 0,Y 488.427,Z 549.53,A -85,B 0,C 180,E1 6349.8,E2 6349.8} C_VEL
LIN {X 0,Y 487.982,Z 552.339,A -85,B 0,C 180,E1 6350.997,E2 6350.997} C_VEL
LIN {X 0,Y 487.801,Z 560.527,A -85,B 0,C 180,E1 6352.175,E2 6352.175} C_VEL
LIN {X 0,Y 489.745,Z 569.518,A -85,B 0,C 180,E1 6352.835,E2 6352.835} C_VEL
LIN {X 0,Y 500.904,Z 591.763,A -85,B 0,C 180,E1 6354.066,E2 6354.066} C_VEL
LIN {X 0,Y 499.693,Z 634.485,A -85,B 0,C 180,E1 6355.037,E2 6355.037} C_VEL
LIN {X 0,Y 497.178,Z 674.236,A -85,B 0,C 180,E1 6356.638,E2 6356.638} C_VEL
LIN {X 0,Y 494.007,Z 712.733,A -85,B 0,C 180,E1 6358.973,E2 6358.973} C_VEL
LIN {X 0,Y 490.514,Z 745.855,A -85,B 0,C 180,E1 6361.803,E2 6361.803} C_VEL
LIN {X 0,Y 487.249,Z 776.375,A -85,B 0,C 180,E1 6365.287,E2 6365.287} C_VEL
LIN {X 0,Y 484.637,Z 802.501,A -85,B 0,C 180,E1 6369.223,E2 6369.223} C_VEL
LIN {X 0,Y 482.858,Z 822.881,A -85,B 0,C 180,E1 6373.277,E2 6373.277} C_VEL
LIN {X 0,Y 481.915,Z 839.405,A -85,B 0,C 180,E1 6377.799,E2 6377.799} C_VEL
LIN {X 0,Y 481.565,Z 849.598,A -85,B 0,C 180,E1 6381.895,E2 6381.895} C_VEL
LIN {X 0,Y 481.404,Z 855.91,A -85,B 0,C 180,E1 6386.407,E2 6386.407} C_VEL
LIN {X 0,Y 481.441,Z 857.5,A -85,B 0,C 180,E1 6390.001,E2 6390.001} C_VEL
LIN {X 0,Y 481.402,Z 855.909,A -85,B 0,C 180,E1 6393.596,E2 6393.596} C_VEL
LIN {X 0,Y 481.587,Z 849.594,A -85,B 0,C 180,E1 6398.107,E2 6398.107} C_VEL
LIN {X 0,Y 482.137,Z 836.852,A -85,B 0,C 180,E1 6403.014,E2 6403.014} C_VEL
LIN {X 0,Y 483.253,Z 819.453,A -85,B 0,C 180,E1 6407.485,E2 6407.485} C_VEL
LIN {X 0,Y 485.162,Z 797.433,A -85,B 0,C 180,E1 6411.629,E2 6411.629} C_VEL
LIN {X 0,Y 487.825,Z 770.844,A -85,B 0,C 180,E1 6415.418,E2 6415.418} C_VEL
LIN {X 0,Y 491.033,Z 740.59,A -85,B 0,C 180,E1 6418.705,E2 6418.705} C_VEL
LIN {X 0,Y 494.396,Z 707.655,A -85,B 0,C 180,E1 6421.387,E2 6421.387} C_VEL
LIN {X 0,Y 497.449,Z 669.904,A -85,B 0,C 180,E1 6423.581,E2 6423.581} C_VEL
LIN {X 0,Y 499.887,Z 630.375,A -85,B 0,C 180,E1 6425.101,E2 6425.101} C_VEL
LIN {X 0,Y 500.618,Z 591.648,A -85,B 0,C 180,E1 6425.981,E2 6425.981} C_VEL
LIN {X 0,Y 480.698,Z 551.04,A -85,B 0,C 180,E1 6428.291,E2 6428.291} C_VEL
LIN {X 0,Y 480.562,Z 549.53,A -85,B 0,C 180,E1 6428.382,E2 6428.382} C_VEL
LIN {X 0,Y 480.469,Z 549.53,A -85,B 0,C 180,E1 6433.743,E2 6433.743} C_VEL
LIN {X 0,Y 480.504,Z 549.53,A -85,B 0,C 180,E1 6438.915,E2 6438.915} C_VEL
LIN {X 0,Y 480.465,Z 549.53,A -85,B 0,C 180,E1 6444.747,E2 6444.747} C_VEL
LIN {X 0,Y 480.505,Z 549.53,A -85,B 0,C 180,E1 6449.827,E2 6449.827} C_VEL
LIN {X 0,Y 480.626,Z 549.53,A -85,B 0,C 180,E1 6455.9,E2 6455.9} C_VEL
LIN {X 0,Y 480.873,Z 549.53,A -85,B 0,C 180,E1 6461.7,E2 6461.7} C_VEL
LIN {X 0,Y 480.79,Z 549.53,A -85,B 0,C 180,E1 6467.296,E2 6467.296} C_VEL
LIN {X 0,Y 481.136,Z 549.53,A -85,B 0,C 180,E1 6472.78,E2 6472.78} C_VEL
LIN {X 0,Y 481.438,Z 549.53,A -85,B 0,C 180,E1 6478.189,E2 6478.189} C_VEL
LIN {X 0,Y 481.305,Z 549.53,A -85,B 0,C 180,E1 6483.579,E2 6483.579} C_VEL
LIN {X 0,Y 481.093,Z 549.53,A -85,B 0,C 180,E1 6489.006,E2 6489.006} C_VEL
LIN {X 0,Y 480.998,Z 549.53,A -85,B 0,C 180,E1 6494.517,E2 6494.517} C_VEL
LIN {X 0,Y 480.814,Z 549.53,A -85,B 0,C 180,E1 6500.175,E2 6500.175} C_VEL
LIN {X 0,Y 480.643,Z 549.53,A -85,B 0,C 180,E1 6506.051,E2 6506.051} C_VEL
LIN {X 0,Y 480.677,Z 549.53,A -85,B 0,C 180,E1 6512.229,E2 6512.229} C_VEL
LIN {X 0,Y 480.623,Z 549.53,A -85,B 0,C 180,E1 6518.284,E2 6518.284} C_VEL
LIN {X 0,Y 480.429,Z 549.53,A -85,B 0,C 180,E1 6523.743,E2 6523.743} C_VEL
LIN {X 0,Y 480.502,Z 549.53,A -85,B 0,C 180,E1 6528.875,E2 6528.875} C_VEL
LIN {X 0,Y 480.635,Z 549.53,A -85,B 0,C 180,E1 6534.671,E2 6534.671} C_VEL
LIN {X 0,Y 480.651,Z 549.53,A -85,B 0,C 180,E1 6539.845,E2 6539.845} C_VEL
LIN {X 0,Y 480.652,Z 549.53,A -85,B 0,C 180,E1 6545.911,E2 6545.911} C_VEL
LIN {X 0,Y 480.808,Z 549.53,A -85,B 0,C 180,E1 6551.707,E2 6551.707} C_VEL
LIN {X 0,Y 480.953,Z 549.53,A -85,B 0,C 180,E1 6557.311,E2 6557.311} C_VEL
LIN {X 0,Y 481.072,Z 549.53,A -85,B 0,C 180,E1 6563.402,E2 6563.402} C_VEL
LIN {X 0,Y 495.93,Z 586.27,A -85,B 0,C 180,E1 6565.542,E2 6565.542} C_VEL
LIN {X 0,Y 493.831,Z 623.644,A -85,B 0,C 180,E1 6567.152,E2 6567.152} C_VEL
LIN {X 0,Y 491.103,Z 656.408,A -85,B 0,C 180,E1 6569.271,E2 6569.271} C_VEL
LIN {X 0,Y 488.171,Z 687.677,A -85,B 0,C 180,E1 6572.102,E2 6572.102} C_VEL
LIN {X 0,Y 485.428,Z 715.37,A -85,B 0,C 180,E1 6575.549,E2 6575.549} C_VEL
LIN {X 0,Y 483.459,Z 737.722,A -85,B 0,C 180,E1 6579.346,E2 6579.346} C_VEL
LIN {X 0,Y 482.149,Z 756.446,A -85,B 0,C 180,E1 6583.72,E2 6583.72} C_VEL
LIN {X 0,Y 481.669,Z 767.71,A -85,B 0,C 180,E1 6587.549,E2 6587.549} C_VEL
LIN {X 0,Y 481.353,Z 774.252,A -85,B 0,C 180,E1 6591.131,E2 6591.131} C_VEL
LIN {X 0,Y 481.002,Z 777.244,A -85,B 0,C 180,E1 6594.588,E2 6594.588} C_VEL
LIN {X 0,Y 481.12,Z 776.511,A -85,B 0,C 180,E1 6598.629,E2 6598.629} C_VEL
LIN {X 0,Y 481.487,Z 771.994,A -85,B 0,C 180,E1 6602.249,E2 6602.249} C_VEL
LIN {X 0,Y 481.843,Z 761.904,A -85,B 0,C 180,E1 6606.513,E2 6606.513} C_VEL
LIN {X 0,Y 482.711,Z 746.377,A -85,B 0,C 180,E1 6610.723,E2 6610.723} C_VEL
LIN {X 0,Y 484.389,Z 726.083,A -85,B 0,C 180,E1 6614.712,E2 6614.712} C_VEL
LIN {X 0,Y 486.82,Z 701.558,A -85,B 0,C 180,E1 6618.241,E2 6618.241} C_VEL
LIN {X 0,Y 489.823,Z 671.995,A -85,B 0,C 180,E1 6621.381,E2 6621.381} C_VEL
LIN {X 0,Y 492.894,Z 638.482,A -85,B 0,C 180,E1 6623.927,E2 6623.927} C_VEL
LIN {X 0,Y 495.343,Z 604.943,A -85,B 0,C 180,E1 6625.686,E2 6625.686} C_VEL
LIN {X 0,Y 495.685,Z 585.433,A -85,B 0,C 180,E1 6626.466,E2 6626.466} C_VEL
LIN {X 0,Y 480.544,Z 549.53,A -85,B 0,C 180,E1 6628.622,E2 6628.622} C_VEL
LIN {X 0,Y 480.608,Z 549.53,A -85,B 0,C 180,E1 6633.947,E2 6633.947} C_VEL
LIN {X 0,Y 480.9,Z 549.53,A -85,B 0,C 180,E1 6640.278,E2 6640.278} C_VEL
LIN {X 0,Y 480.734,Z 549.53,A -85,B 0,C 180,E1 6646.67,E2 6646.67} C_VEL
LIN {X 0,Y 481.13,Z 549.53,A -85,B 0,C 180,E1 6653.008,E2 6653.008} C_VEL
LIN {X 0,Y 481.417,Z 549.53,A -85,B 0,C 180,E1 6658.219,E2 6658.219} C_VEL
LIN {X 0,Y 481.297,Z 549.53,A -85,B 0,C 180,E1 6663.609,E2 6663.609} C_VEL
LIN {X 0,Y 481.104,Z 549.53,A -85,B 0,C 180,E1 6669.036,E2 6669.036} C_VEL
LIN {X 0,Y 480.986,Z 549.53,A -85,B 0,C 180,E1 6674.548,E2 6674.548} C_VEL
LIN {X 0,Y 480.841,Z 549.53,A -85,B 0,C 180,E1 6680.206,E2 6680.206} C_VEL
LIN {X 0,Y 480.661,Z 549.53,A -85,B 0,C 180,E1 6686.084,E2 6686.084} C_VEL
LIN {X 0,Y 480.677,Z 549.53,A -85,B 0,C 180,E1 6692.264,E2 6692.264} C_VEL
LIN {X 0,Y 480.6,Z 549.53,A -85,B 0,C 180,E1 6698.285,E2 6698.285} C_VEL
LIN {X 0,Y 480.408,Z 549.53,A -85,B 0,C 180,E1 6703.745,E2 6703.745} C_VEL
LIN {X 0,Y 480.438,Z 549.53,A -85,B 0,C 180,E1 6709.802,E2 6709.802} C_VEL
LIN {X 0,Y 480.634,Z 549.53,A -85,B 0,C 180,E1 6711.719,E2 6711.719} C_VEL
LIN {X 0,Y 489.745,Z 569.518,A -85,B 0,C 180,E1 6712.835,E2 6712.835} C_VEL
LIN {X 0,Y 493.542,Z 586.039,A -85,B 0,C 180,E1 6713.412,E2 6713.412} C_VEL
LIN {X 0,Y 494.164,Z 603.557,A -85,B 0,C 180,E1 6713.783,E2 6713.783} C_VEL
LIN {X 0,Y 492.314,Z 643.442,A -85,B 0,C 180,E1 6714.855,E2 6714.855} C_VEL
LIN {X 0,Y 489.547,Z 682.614,A -85,B 0,C 180,E1 6716.633,E2 6716.633} C_VEL
LIN {X 0,Y 486.074,Z 719.917,A -85,B 0,C 180,E1 6719.091,E2 6719.091} C_VEL
LIN {X 0,Y 482.512,Z 753.787,A -85,B 0,C 180,E1 6722.171,E2 6722.171} C_VEL
LIN {X 0,Y 478.947,Z 784.662,A -85,B 0,C 180,E1 6726.028,E2 6726.028} C_VEL
LIN {X 0,Y 476.32,Z 810.345,A -85,B 0,C 180,E1 6730.331,E2 6730.331} C_VEL
LIN {X 0,Y 474.692,Z 830.028,A -85,B 0,C 180,E1 6734.797,E2 6734.797} C_VEL
LIN {X 0,Y 473.928,Z 844.453,A -85,B 0,C 180,E1 6739.452,E2 6739.452} C_VEL
LIN {X 0,Y 473.651,Z 852.752,A -85,B 0,C 180,E1 6743.599,E2 6743.599} C_VEL
LIN {X 0,Y 473.535,Z 857.09,A -85,B 0,C 180,E1 6748.175,E2 6748.175} C_VEL
LIN {X 0,Y 473.601,Z 857.089,A -85,B 0,C 180,E1 6751.827,E2 6751.827} C_VEL
LIN {X 0,Y 473.651,Z 852.752,A -85,B 0,C 180,E1 6756.404,E2 6756.404} C_VEL
LIN {X 0,Y 473.878,Z 843.302,A -85,B 0,C 180,E1 6761.016,E2 6761.016} C_VEL
LIN {X 0,Y 474.83,Z 828.285,A -85,B 0,C 180,E1 6765.673,E2 6765.673} C_VEL
LIN {X 0,Y 476.662,Z 806.644,A -85,B 0,C 180,E1 6770.381,E2 6770.381} C_VEL
LIN {X 0,Y 479.341,Z 781.592,A -85,B 0,C 180,E1 6774.407,E2 6774.407} C_VEL
LIN {X 0,Y 482.791,Z 750.989,A -85,B 0,C 180,E1 6778.121,E2 6778.121} C_VEL
LIN {X 0,Y 486.15,Z 718.868,A -85,B 0,C 180,E1 6780.999,E2 6780.999} C_VEL
LIN {X 0,Y 489.649,Z 681.832,A -85,B 0,C 180,E1 6783.429,E2 6783.429} C_VEL
LIN {X 0,Y 492.434,Z 643.43,A -85,B 0,C 180,E1 6785.165,E2 6785.165} C_VEL
LIN {X 0,Y 494.453,Z 604.901,A -85,B 0,C 180,E1 6786.2,E2 6786.2} C_VEL
LIN {X 0,Y 493.819,Z 593.671,A -85,B 0,C 180,E1 6786.469,E2 6786.469} C_VEL
LIN {X 0,Y 472.611,Z 549.53,A -85,B 0,C 180,E1 6789.131,E2 6789.131} C_VEL
LIN {X 0,Y 472.507,Z 549.53,A -85,B 0,C 180,E1 6795.356,E2 6795.356} C_VEL
LIN {X 0,Y 472.547,Z 549.53,A -85,B 0,C 180,E1 6800.299,E2 6800.299} C_VEL
LIN {X 0,Y 472.533,Z 549.53,A -85,B 0,C 180,E1 6806.132,E2 6806.132} C_VEL
LIN {X 0,Y 472.594,Z 549.53,A -85,B 0,C 180,E1 6811.373,E2 6811.373} C_VEL
LIN {X 0,Y 472.832,Z 549.53,A -85,B 0,C 180,E1 6817.75,E2 6817.75} C_VEL
LIN {X 0,Y 472.927,Z 549.53,A -85,B 0,C 180,E1 6823.299,E2 6823.299} C_VEL
LIN {X 0,Y 472.98,Z 549.53,A -85,B 0,C 180,E1 6828.951,E2 6828.951} C_VEL
LIN {X 0,Y 473.276,Z 549.53,A -85,B 0,C 180,E1 6834.497,E2 6834.497} C_VEL
LIN {X 0,Y 473.381,Z 549.53,A -85,B 0,C 180,E1 6839.985,E2 6839.985} C_VEL
LIN {X 0,Y 473.248,Z 549.53,A -85,B 0,C 180,E1 6845.473,E2 6845.473} C_VEL
LIN {X 0,Y 473.108,Z 549.53,A -85,B 0,C 180,E1 6851.015,E2 6851.015} C_VEL
LIN {X 0,Y 472.957,Z 549.53,A -85,B 0,C 180,E1 6856.823,E2 6856.823} C_VEL
LIN {X 0,Y 472.837,Z 549.53,A -85,B 0,C 180,E1 6862.496,E2 6862.496} C_VEL
LIN {X 0,Y 472.702,Z 549.53,A -85,B 0,C 180,E1 6868.585,E2 6868.585} C_VEL
LIN {X 0,Y 472.743,Z 549.53,A -85,B 0,C 180,E1 6875.041,E2 6875.041} C_VEL
LIN {X 0,Y 472.552,Z 549.53,A -85,B 0,C 180,E1 6879.966,E2 6879.966} C_VEL
LIN {X 0,Y 472.443,Z 549.53,A -85,B 0,C 180,E1 6885.355,E2 6885.355} C_VEL
LIN {X 0,Y 472.568,Z 549.53,A -85,B 0,C 180,E1 6890.307,E2 6890.307} C_VEL
LIN {X 0,Y 472.701,Z 549.53,A -85,B 0,C 180,E1 6896.052,E2 6896.052} C_VEL
LIN {X 0,Y 472.68,Z 549.53,A -85,B 0,C 180,E1 6901.387,E2 6901.387} C_VEL
LIN {X 0,Y 472.838,Z 549.53,A -85,B 0,C 180,E1 6907.672,E2 6907.672} C_VEL
LIN {X 0,Y 472.939,Z 549.53,A -85,B 0,C 180,E1 6913.31,E2 6913.31} C_VEL
LIN {X 0,Y 473.082,Z 549.53,A -85,B 0,C 180,E1 6918.965,E2 6918.965} C_VEL
LIN {X 0,Y 473.191,Z 549.53,A -85,B 0,C 180,E1 6922.763,E2 6922.763} C_VEL
LIN {X 0,Y 488.862,Z 587.603,A -85,B 0,C 180,E1 6925.059,E2 6925.059} C_VEL
LIN {X 0,Y 487,Z 623.805,A -85,B 0,C 180,E1 6926.668,E2 6926.668} C_VEL
LIN {X 0,Y 483.967,Z 658.209,A -85,B 0,C 180,E1 6928.933,E2 6928.933} C_VEL
LIN {X 0,Y 480.849,Z 689.128,A -85,B 0,C 180,E1 6931.797,E2 6931.797} C_VEL
LIN {X 0,Y 477.961,Z 716.005,A -85,B 0,C 180,E1 6935.206,E2 6935.206} C_VEL
LIN {X 0,Y 475.826,Z 738.656,A -85,B 0,C 180,E1 6939.122,E2 6939.122} C_VEL
LIN {X 0,Y 474.346,Z 756.825,A -85,B 0,C 180,E1 6943.527,E2 6943.527} C_VEL
LIN {X 0,Y 473.748,Z 768.711,A -85,B 0,C 180,E1 6947.864,E2 6947.864} C_VEL
LIN {X 0,Y 473.422,Z 774.816,A -85,B 0,C 180,E1 6951.479,E2 6951.479} C_VEL
LIN {X 0,Y 473.116,Z 777.217,A -85,B 0,C 180,E1 6954.495,E2 6954.495} C_VEL
LIN {X 0,Y 473.261,Z 776.108,A -85,B 0,C 180,E1 6959.15,E2 6959.15} C_VEL
LIN {X 0,Y 473.73,Z 769.919,A -85,B 0,C 180,E1 6963.467,E2 6963.467} C_VEL
LIN {X 0,Y 474.408,Z 757.192,A -85,B 0,C 180,E1 6968.276,E2 6968.276} C_VEL
LIN {X 0,Y 475.644,Z 740.25,A -85,B 0,C 180,E1 6972.495,E2 6972.495} C_VEL
LIN {X 0,Y 477.782,Z 718.304,A -85,B 0,C 180,E1 6976.394,E2 6976.394} C_VEL
LIN {X 0,Y 480.676,Z 691.999,A -85,B 0,C 180,E1 6979.834,E2 6979.834} C_VEL
LIN {X 0,Y 483.95,Z 660.238,A -85,B 0,C 180,E1 6982.867,E2 6982.867} C_VEL
LIN {X 0,Y 487.083,Z 626.011,A -85,B 0,C 180,E1 6985.165,E2 6985.165} C_VEL
LIN {X 0,Y 489.078,Z 588.133,A -85,B 0,C 180,E1 6986.881,E2 6986.881} C_VEL
LIN {X 0,Y 474.188,Z 554.246,A -85,B 0,C 180,E1 6989.059,E2 6989.059} C_VEL
LIN {X 0,Y 472.594,Z 549.53,A -85,B 0,C 180,E1 6989.303,E2 6989.303} C_VEL
LIN {X 0,Y 472.741,Z 549.53,A -85,B 0,C 180,E1 6995.506,E2 6995.506} C_VEL
LIN {X 0,Y 472.973,Z 549.53,A -85,B 0,C 180,E1 7001.415,E2 7001.415} C_VEL
LIN {X 0,Y 472.896,Z 549.53,A -85,B 0,C 180,E1 7007.112,E2 7007.112} C_VEL
LIN {X 0,Y 473.198,Z 549.53,A -85,B 0,C 180,E1 7013.002,E2 7013.002} C_VEL
LIN {X 0,Y 473.507,Z 549.53,A -85,B 0,C 180,E1 7018.189,E2 7018.189} C_VEL
LIN {X 0,Y 473.384,Z 549.53,A -85,B 0,C 180,E1 7023.67,E2 7023.67} C_VEL
LIN {X 0,Y 473.208,Z 549.53,A -85,B 0,C 180,E1 7029.188,E2 7029.188} C_VEL
LIN {X 0,Y 473.047,Z 549.53,A -85,B 0,C 180,E1 7034.798,E2 7034.798} C_VEL
LIN {X 0,Y 472.891,Z 549.53,A -85,B 0,C 180,E1 7040.561,E2 7040.561} C_VEL
LIN {X 0,Y 472.715,Z 549.53,A -85,B 0,C 180,E1 7046.645,E2 7046.645} C_VEL
LIN {X 0,Y 472.696,Z 549.53,A -85,B 0,C 180,E1 7052.877,E2 7052.877} C_VEL
LIN {X 0,Y 472.693,Z 549.53,A -85,B 0,C 180,E1 7057.349,E2 7057.349} C_VEL
LIN {X 0,Y 472.45,Z 549.53,A -85,B 0,C 180,E1 7062.727,E2 7062.727} C_VEL
LIN {X 0,Y 472.449,Z 549.53,A -85,B 0,C 180,E1 7067.877,E2 7067.877} C_VEL
LIN {X 0,Y 472.68,Z 549.633,A -85,B 0,C 180,E1 7071.062,E2 7071.062} C_VEL
LIN {X 0,Y 494.359,Z 595.228,A -85,B 0,C 180,E1 7073.633,E2 7073.633} C_VEL
LIN {X 0,Y 494.164,Z 603.557,A -85,B 0,C 180,E1 7073.783,E2 7073.783} C_VEL
LIN {X 0,Y 490.3,Z 620.651,A -85,B 0,C 180,E1 7073.907,E2 7073.907} C_VEL
LIN {X 0,Y 486.051,Z 637.478,A -85,B 0,C 180,E1 7074.163,E2 7074.163} C_VEL
LIN {X 0,Y 483.218,Z 675.769,A -85,B 0,C 180,E1 7075.8,E2 7075.8} C_VEL
LIN {X 0,Y 479.864,Z 711.371,A -85,B 0,C 180,E1 7078.025,E2 7078.025} C_VEL
LIN {X 0,Y 475.935,Z 746.669,A -85,B 0,C 180,E1 7081.051,E2 7081.051} C_VEL
LIN {X 0,Y 472.747,Z 774.626,A -85,B 0,C 180,E1 7084.222,E2 7084.222} C_VEL
LIN {X 0,Y 469.537,Z 801.768,A -85,B 0,C 180,E1 7088.385,E2 7088.385} C_VEL
LIN {X 0,Y 467.365,Z 823.418,A -85,B 0,C 180,E1 7092.84,E2 7092.84} C_VEL
LIN {X 0,Y 466.212,Z 839.405,A -85,B 0,C 180,E1 7097.382,E2 7097.382} C_VEL
LIN {X 0,Y 465.818,Z 849.893,A -85,B 0,C 180,E1 7101.766,E2 7101.766} C_VEL
LIN {X 0,Y 465.619,Z 855.91,A -85,B 0,C 180,E1 7106.285,E2 7106.285} C_VEL
LIN {X 0,Y 465.654,Z 857.5,A -85,B 0,C 180,E1 7110.001,E2 7110.001} C_VEL
LIN {X 0,Y 465.624,Z 855.91,A -85,B 0,C 180,E1 7113.718,E2 7113.718} C_VEL
LIN {X 0,Y 465.841,Z 849.871,A -85,B 0,C 180,E1 7118.247,E2 7118.247} C_VEL
LIN {X 0,Y 466.401,Z 838.037,A -85,B 0,C 180,E1 7123.091,E2 7123.091} C_VEL
LIN {X 0,Y 467.734,Z 820.003,A -85,B 0,C 180,E1 7127.96,E2 7127.96} C_VEL
LIN {X 0,Y 470.108,Z 797.05,A -85,B 0,C 180,E1 7132.424,E2 7132.424} C_VEL
LIN {X 0,Y 473.173,Z 770.832,A -85,B 0,C 180,E1 7136.265,E2 7136.265} C_VEL
LIN {X 0,Y 476.765,Z 739.482,A -85,B 0,C 180,E1 7139.654,E2 7139.654} C_VEL
LIN {X 0,Y 480.473,Z 705.76,A -85,B 0,C 180,E1 7142.397,E2 7142.397} C_VEL
LIN {X 0,Y 483.944,Z 668.045,A -85,B 0,C 180,E1 7144.619,E2 7144.619} C_VEL
LIN {X 0,Y 486.615,Z 630.097,A -85,B 0,C 180,E1 7146.102,E2 7146.102} C_VEL
LIN {X 0,Y 487.457,Z 596.894,A -85,B 0,C 180,E1 7146.914,E2 7146.914} C_VEL
LIN {X 0,Y 464.769,Z 550.818,A -85,B 0,C 180,E1 7149.717,E2 7149.717} C_VEL
LIN {X 0,Y 464.651,Z 549.53,A -85,B 0,C 180,E1 7149.851,E2 7149.851} C_VEL
LIN {X 0,Y 464.582,Z 549.53,A -85,B 0,C 180,E1 7155.611,E2 7155.611} C_VEL
LIN {X 0,Y 464.617,Z 549.53,A -85,B 0,C 180,E1 7161.887,E2 7161.887} C_VEL
LIN {X 0,Y 464.578,Z 549.53,A -85,B 0,C 180,E1 7168.678,E2 7168.678} C_VEL
LIN {X 0,Y 464.823,Z 549.53,A -85,B 0,C 180,E1 7175.371,E2 7175.371} C_VEL
LIN {X 0,Y 464.996,Z 549.53,A -85,B 0,C 180,E1 7181.052,E2 7181.052} C_VEL
LIN {X 0,Y 464.948,Z 549.53,A -85,B 0,C 180,E1 7186.856,E2 7186.856} C_VEL
LIN {X 0,Y 465.308,Z 549.53,A -85,B 0,C 180,E1 7192.533,E2 7192.533} C_VEL
LIN {X 0,Y 465.625,Z 549.53,A -85,B 0,C 180,E1 7198.128,E2 7198.128} C_VEL
LIN {X 0,Y 465.491,Z 549.53,A -85,B 0,C 180,E1 7203.701,E2 7203.701} C_VEL
LIN {X 0,Y 465.268,Z 549.53,A -85,B 0,C 180,E1 7209.315,E2 7209.315} C_VEL
LIN {X 0,Y 465.135,Z 549.53,A -85,B 0,C 180,E1 7215.023,E2 7215.023} C_VEL
LIN {X 0,Y 464.945,Z 549.53,A -85,B 0,C 180,E1 7220.895,E2 7220.895} C_VEL
LIN {X 0,Y 464.77,Z 549.53,A -85,B 0,C 180,E1 7227.012,E2 7227.012} C_VEL
LIN {X 0,Y 464.782,Z 549.53,A -85,B 0,C 180,E1 7233.473,E2 7233.473} C_VEL
LIN {X 0,Y 464.66,Z 549.53,A -85,B 0,C 180,E1 7238.791,E2 7238.791} C_VEL
LIN {X 0,Y 464.549,Z 549.53,A -85,B 0,C 180,E1 7245.577,E2 7245.577} C_VEL
LIN {X 0,Y 464.674,Z 549.53,A -85,B 0,C 180,E1 7251.9,E2 7251.9} C_VEL
LIN {X 0,Y 464.752,Z 549.53,A -85,B 0,C 180,E1 7257.536,E2 7257.536} C_VEL
LIN {X 0,Y 464.738,Z 549.53,A -85,B 0,C 180,E1 7262.96,E2 7262.96} C_VEL
LIN {X 0,Y 464.903,Z 549.53,A -85,B 0,C 180,E1 7269.08,E2 7269.08} C_VEL
LIN {X 0,Y 465.109,Z 549.53,A -85,B 0,C 180,E1 7274.955,E2 7274.955} C_VEL
LIN {X 0,Y 465.241,Z 549.53,A -85,B 0,C 180,E1 7280.665,E2 7280.665} C_VEL
LIN {X 0,Y 465.232,Z 549.696,A -85,B 0,C 180,E1 7282.098,E2 7282.098} C_VEL
LIN {X 0,Y 481.716,Z 588.627,A -85,B 0,C 180,E1 7284.544,E2 7284.544} C_VEL
LIN {X 0,Y 482.32,Z 597.253,A -85,B 0,C 180,E1 7284.946,E2 7284.946} C_VEL
LIN {X 0,Y 479.67,Z 631.77,A -85,B 0,C 180,E1 7286.617,E2 7286.617} C_VEL
LIN {X 0,Y 476.343,Z 664.964,A -85,B 0,C 180,E1 7288.997,E2 7288.997} C_VEL
LIN {X 0,Y 472.956,Z 695.496,A -85,B 0,C 180,E1 7292.056,E2 7292.056} C_VEL
LIN {X 0,Y 469.927,Z 722.471,A -85,B 0,C 180,E1 7295.756,E2 7295.756} C_VEL
LIN {X 0,Y 467.694,Z 744.143,A -85,B 0,C 180,E1 7299.87,E2 7299.87} C_VEL
LIN {X 0,Y 466.374,Z 759.736,A -85,B 0,C 180,E1 7304.025,E2 7304.025} C_VEL
LIN {X 0,Y 465.833,Z 770.256,A -85,B 0,C 180,E1 7308.238,E2 7308.238} C_VEL
LIN {X 0,Y 465.29,Z 776.529,A -85,B 0,C 180,E1 7312.902,E2 7312.902} C_VEL
LIN {X 0,Y 465.185,Z 777.516,A -85,B 0,C 180,E1 7317.008,E2 7317.008} C_VEL
LIN {X 0,Y 465.636,Z 774.215,A -85,B 0,C 180,E1 7321.231,E2 7321.231} C_VEL
LIN {X 0,Y 466.082,Z 766.011,A -85,B 0,C 180,E1 7325.644,E2 7325.644} C_VEL
LIN {X 0,Y 467.029,Z 751.69,A -85,B 0,C 180,E1 7330.255,E2 7330.255} C_VEL
LIN {X 0,Y 468.82,Z 732.44,A -85,B 0,C 180,E1 7334.475,E2 7334.475} C_VEL
LIN {X 0,Y 471.629,Z 707.773,A -85,B 0,C 180,E1 7338.379,E2 7338.379} C_VEL
LIN {X 0,Y 475.114,Z 678.211,A -85,B 0,C 180,E1 7341.763,E2 7341.763} C_VEL
LIN {X 0,Y 478.448,Z 647.174,A -85,B 0,C 180,E1 7344.347,E2 7344.347} C_VEL
LIN {X 0,Y 481.516,Z 612.416,A -85,B 0,C 180,E1 7346.378,E2 7346.378} C_VEL
LIN {X 0,Y 482.223,Z 590.127,A -85,B 0,C 180,E1 7347.347,E2 7347.347} C_VEL
LIN {X 0,Y 466.702,Z 554.801,A -85,B 0,C 180,E1 7349.71,E2 7349.71} C_VEL
LIN {X 0,Y 464.675,Z 549.53,A -85,B 0,C 180,E1 7350.079,E2 7350.079} C_VEL
LIN {X 0,Y 464.84,Z 549.53,A -85,B 0,C 180,E1 7355.359,E2 7355.359} C_VEL
LIN {X 0,Y 465.023,Z 549.53,A -85,B 0,C 180,E1 7361.086,E2 7361.086} C_VEL
LIN {X 0,Y 464.994,Z 549.53,A -85,B 0,C 180,E1 7366.889,E2 7366.889} C_VEL
LIN {X 0,Y 465.288,Z 549.53,A -85,B 0,C 180,E1 7372.998,E2 7372.998} C_VEL
LIN {X 0,Y 465.604,Z 549.53,A -85,B 0,C 180,E1 7378.159,E2 7378.159} C_VEL
LIN {X 0,Y 465.484,Z 549.53,A -85,B 0,C 180,E1 7383.732,E2 7383.732} C_VEL
LIN {X 0,Y 465.281,Z 549.53,A -85,B 0,C 180,E1 7389.346,E2 7389.346} C_VEL
LIN {X 0,Y 465.106,Z 549.53,A -85,B 0,C 180,E1 7395.056,E2 7395.056} C_VEL
LIN {X 0,Y 464.973,Z 549.53,A -85,B 0,C 180,E1 7400.927,E2 7400.927} C_VEL
LIN {X 0,Y 464.787,Z 549.53,A -85,B 0,C 180,E1 7407.045,E2 7407.045} C_VEL
LIN {X 0,Y 464.779,Z 549.53,A -85,B 0,C 180,E1 7413.51,E2 7413.51} C_VEL
LIN {X 0,Y 464.616,Z 549.53,A -85,B 0,C 180,E1 7418.788,E2 7418.788} C_VEL
LIN {X 0,Y 464.507,Z 549.53,A -85,B 0,C 180,E1 7425.627,E2 7425.627} C_VEL
LIN {X 0,Y 464.693,Z 550.121,A -85,B 0,C 180,E1 7430.354,E2 7430.354} C_VEL
LIN {X 0,Y 487.73,Z 598.623,A -85,B 0,C 180,E1 7433.188,E2 7433.188} C_VEL
LIN {X 0,Y 486.051,Z 637.478,A -85,B 0,C 180,E1 7434.163,E2 7434.163} C_VEL
LIN {X 0,Y 477.099,Z 668.459,A -85,B 0,C 180,E1 7434.953,E2 7434.953} C_VEL
LIN {X 0,Y 476.856,Z 670.428,A -85,B 0,C 180,E1 7435.043,E2 7435.043} C_VEL
LIN {X 0,Y 472.96,Z 709.206,A -85,B 0,C 180,E1 7437.415,E2 7437.415} C_VEL
LIN {X 0,Y 468.854,Z 744.66,A -85,B 0,C 180,E1 7440.459,E2 7440.459} C_VEL
LIN {X 0,Y 465.113,Z 775.744,A -85,B 0,C 180,E1 7444.026,E2 7444.026} C_VEL
LIN {X 0,Y 462.244,Z 800.045,A -85,B 0,C 180,E1 7447.699,E2 7447.699} C_VEL
LIN {X 0,Y 459.852,Z 821.707,A -85,B 0,C 180,E1 7452.118,E2 7452.118} C_VEL
LIN {X 0,Y 458.503,Z 838.043,A -85,B 0,C 180,E1 7456.682,E2 7456.682} C_VEL
LIN {X 0,Y 457.949,Z 849.32,A -85,B 0,C 180,E1 7461.336,E2 7461.336} C_VEL
LIN {X 0,Y 457.712,Z 855.909,A -85,B 0,C 180,E1 7466.221,E2 7466.221} C_VEL
LIN {X 0,Y 457.754,Z 857.5,A -85,B 0,C 180,E1 7470.001,E2 7470.001} C_VEL
LIN {X 0,Y 457.72,Z 855.909,A -85,B 0,C 180,E1 7473.782,E2 7473.782} C_VEL
LIN {X 0,Y 457.969,Z 849.289,A -85,B 0,C 180,E1 7478.681,E2 7478.681} C_VEL
LIN {X 0,Y 458.556,Z 838.036,A -85,B 0,C 180,E1 7483.319,E2 7483.319} C_VEL
LIN {X 0,Y 459.95,Z 820.938,A -85,B 0,C 180,E1 7488.061,E2 7488.061} C_VEL
LIN {X 0,Y 462.438,Z 798.592,A -85,B 0,C 180,E1 7492.547,E2 7492.547} C_VEL
LIN {X 0,Y 465.57,Z 772.036,A -85,B 0,C 180,E1 7496.468,E2 7496.468} C_VEL
LIN {X 0,Y 469.48,Z 739.886,A -85,B 0,C 180,E1 7500.029,E2 7500.029} C_VEL
LIN {X 0,Y 473.54,Z 704.886,A -85,B 0,C 180,E1 7502.92,E2 7502.92} C_VEL
LIN {X 0,Y 477.224,Z 667.289,A -85,B 0,C 180,E1 7505.152,E2 7505.152} C_VEL
LIN {X 0,Y 480.132,Z 628.427,A -85,B 0,C 180,E1 7506.668,E2 7506.668} C_VEL
LIN {X 0,Y 480.793,Z 599.221,A -85,B 0,C 180,E1 7507.409,E2 7507.409} C_VEL
LIN {X 0,Y 456.801,Z 550.93,A -85,B 0,C 180,E1 7510.473,E2 7510.473} C_VEL
LIN {X 0,Y 456.678,Z 549.53,A -85,B 0,C 180,E1 7510.528,E2 7510.528} C_VEL
LIN {X 0,Y 456.709,Z 549.53,A -85,B 0,C 180,E1 7516.629,E2 7516.629} C_VEL
LIN {X 0,Y 456.658,Z 549.53,A -85,B 0,C 180,E1 7523.492,E2 7523.492} C_VEL
LIN {X 0,Y 456.672,Z 549.53,A -85,B 0,C 180,E1 7530.277,E2 7530.277} C_VEL
LIN {X 0,Y 456.891,Z 549.53,A -85,B 0,C 180,E1 7536.639,E2 7536.639} C_VEL
LIN {X 0,Y 457.088,Z 549.53,A -85,B 0,C 180,E1 7543.22,E2 7543.22} C_VEL
LIN {X 0,Y 457.251,Z 549.53,A -85,B 0,C 180,E1 7550.489,E2 7550.489} C_VEL
LIN {X 0,Y 457.506,Z 549.53,A -85,B 0,C 180,E1 7556.203,E2 7556.203} C_VEL
LIN {X 0,Y 457.542,Z 549.53,A -85,B 0,C 180,E1 7561.874,E2 7561.874} C_VEL
LIN {X 0,Y 457.335,Z 549.53,A -85,B 0,C 180,E1 7568.151,E2 7568.151} C_VEL
LIN {X 0,Y 457.278,Z 549.53,A -85,B 0,C 180,E1 7573.337,E2 7573.337} C_VEL
LIN {X 0,Y 457.054,Z 549.53,A -85,B 0,C 180,E1 7579.257,E2 7579.257} C_VEL
LIN {X 0,Y 456.856,Z 549.53,A -85,B 0,C 180,E1 7585.405,E2 7585.405} C_VEL
LIN {X 0,Y 456.826,Z 549.53,A -85,B 0,C 180,E1 7591.879,E2 7591.879} C_VEL
LIN {X 0,Y 456.76,Z 549.53,A -85,B 0,C 180,E1 7598.85,E2 7598.85} C_VEL
LIN {X 0,Y 456.64,Z 549.53,A -85,B 0,C 180,E1 7603.91,E2 7603.91} C_VEL
LIN {X 0,Y 456.713,Z 549.53,A -85,B 0,C 180,E1 7609.419,E2 7609.419} C_VEL
LIN {X 0,Y 456.803,Z 549.53,A -85,B 0,C 180,E1 7615.833,E2 7615.833} C_VEL
LIN {X 0,Y 456.83,Z 549.53,A -85,B 0,C 180,E1 7622.453,E2 7622.453} C_VEL
LIN {X 0,Y 456.947,Z 549.53,A -85,B 0,C 180,E1 7628.698,E2 7628.698} C_VEL
LIN {X 0,Y 457.164,Z 549.53,A -85,B 0,C 180,E1 7634.687,E2 7634.687} C_VEL
LIN {X 0,Y 457.318,Z 549.53,A -85,B 0,C 180,E1 7641.369,E2 7641.369} C_VEL
LIN {X 0,Y 474.581,Z 589.786,A -85,B 0,C 180,E1 7644.019,E2 7644.019} C_VEL
LIN {X 0,Y 475.678,Z 597.396,A -85,B 0,C 180,E1 7644.427,E2 7644.427} C_VEL
LIN {X 0,Y 472.876,Z 631.941,A -85,B 0,C 180,E1 7646.11,E2 7646.11} C_VEL
LIN {X 0,Y 469.433,Z 664.836,A -85,B 0,C 180,E1 7648.485,E2 7648.485} C_VEL
LIN {X 0,Y 465.888,Z 694.879,A -85,B 0,C 180,E1 7651.506,E2 7651.506} C_VEL
LIN {X 0,Y 462.695,Z 720.944,A -85,B 0,C 180,E1 7655.062,E2 7655.062} C_VEL
LIN {X 0,Y 460.257,Z 743.081,A -85,B 0,C 180,E1 7659.196,E2 7659.196} C_VEL
LIN {X 0,Y 458.633,Z 760.332,A -85,B 0,C 180,E1 7663.79,E2 7663.79} C_VEL
LIN {X 0,Y 458.004,Z 771.207,A -85,B 0,C 180,E1 7668.238,E2 7668.238} C_VEL
LIN {X 0,Y 457.466,Z 777.022,A -85,B 0,C 180,E1 7672.613,E2 7672.613} C_VEL
LIN {X 0,Y 457.343,Z 778.115,A -85,B 0,C 180,E1 7677.51,E2 7677.51} C_VEL
LIN {X 0,Y 457.884,Z 774.317,A -85,B 0,C 180,E1 7681.821,E2 7681.821} C_VEL
LIN {X 0,Y 458.347,Z 765.445,A -85,B 0,C 180,E1 7686.341,E2 7686.341} C_VEL
LIN {X 0,Y 459.421,Z 751.568,A -85,B 0,C 180,E1 7690.726,E2 7690.726} C_VEL
LIN {X 0,Y 461.348,Z 732.814,A -85,B 0,C 180,E1 7694.863,E2 7694.863} C_VEL
LIN {X 0,Y 464.274,Z 708.836,A -85,B 0,C 180,E1 7698.715,E2 7698.715} C_VEL
LIN {X 0,Y 467.928,Z 679.874,A -85,B 0,C 180,E1 7702.105,E2 7702.105} C_VEL
LIN {X 0,Y 471.486,Z 648.859,A -85,B 0,C 180,E1 7704.748,E2 7704.748} C_VEL
LIN {X 0,Y 474.682,Z 614.904,A -85,B 0,C 180,E1 7706.788,E2 7706.788} C_VEL
LIN {X 0,Y 475.573,Z 592.679,A -85,B 0,C 180,E1 7707.786,E2 7707.786} C_VEL
LIN {X 0,Y 460.939,Z 559.228,A -85,B 0,C 180,E1 7710.143,E2 7710.143} C_VEL
LIN {X 0,Y 456.765,Z 549.53,A -85,B 0,C 180,E1 7710.781,E2 7710.781} C_VEL
LIN {X 0,Y 456.932,Z 549.53,A -85,B 0,C 180,E1 7717.619,E2 7717.619} C_VEL
LIN {X 0,Y 457.119,Z 549.53,A -85,B 0,C 180,E1 7723.197,E2 7723.197} C_VEL
LIN {X 0,Y 457.121,Z 549.53,A -85,B 0,C 180,E1 7728.595,E2 7728.595} C_VEL
LIN {X 0,Y 457.473,Z 549.53,A -85,B 0,C 180,E1 7734.338,E2 7734.338} C_VEL
LIN {X 0,Y 457.63,Z 549.53,A -85,B 0,C 180,E1 7740.016,E2 7740.016} C_VEL
LIN {X 0,Y 457.441,Z 549.53,A -85,B 0,C 180,E1 7745.694,E2 7745.694} C_VEL
LIN {X 0,Y 457.285,Z 549.53,A -85,B 0,C 180,E1 7751.433,E2 7751.433} C_VEL
LIN {X 0,Y 457.109,Z 549.53,A -85,B 0,C 180,E1 7757.296,E2 7757.296} C_VEL
LIN {X 0,Y 456.934,Z 549.53,A -85,B 0,C 180,E1 7763.358,E2 7763.358} C_VEL
LIN {X 0,Y 456.801,Z 549.53,A -85,B 0,C 180,E1 7769.714,E2 7769.714} C_VEL
LIN {X 0,Y 456.77,Z 549.53,A -85,B 0,C 180,E1 7776.498,E2 7776.498} C_VEL
LIN {X 0,Y 456.613,Z 549.53,A -85,B 0,C 180,E1 7783.362,E2 7783.362} C_VEL
LIN {X 0,Y 456.683,Z 549.53,A -85,B 0,C 180,E1 7789.577,E2 7789.577} C_VEL
LIN {X 0,Y 462.934,Z 562.907,A -85,B 0,C 180,E1 7790.431,E2 7790.431} C_VEL
LIN {X 0,Y 481.108,Z 600.551,A -85,B 0,C 180,E1 7792.701,E2 7792.701} C_VEL
LIN {X 0,Y 479.21,Z 639.534,A -85,B 0,C 180,E1 7793.729,E2 7793.729} C_VEL
LIN {X 0,Y 476.856,Z 670.428,A -85,B 0,C 180,E1 7795.043,E2 7795.043} C_VEL
LIN {X 0,Y 471.905,Z 686.436,A -85,B 0,C 180,E1 7795.672,E2 7795.672} C_VEL
LIN {X 0,Y 466.683,Z 701.928,A -85,B 0,C 180,E1 7796.438,E2 7796.438} C_VEL
LIN {X 0,Y 462.42,Z 737.346,A -85,B 0,C 180,E1 7799.339,E2 7799.339} C_VEL
LIN {X 0,Y 458.408,Z 769.109,A -85,B 0,C 180,E1 7802.833,E2 7802.833} C_VEL
LIN {X 0,Y 455.024,Z 796.573,A -85,B 0,C 180,E1 7806.809,E2 7806.809} C_VEL
LIN {X 0,Y 452.804,Z 816.182,A -85,B 0,C 180,E1 7810.535,E2 7810.535} C_VEL
LIN {X 0,Y 451.005,Z 834.755,A -85,B 0,C 180,E1 7815.394,E2 7815.394} C_VEL
LIN {X 0,Y 450.169,Z 847.681,A -85,B 0,C 180,E1 7820.353,E2 7820.353} C_VEL
LIN {X 0,Y 449.872,Z 853.956,A -85,B 0,C 180,E1 7824.226,E2 7824.226} C_VEL
LIN {X 0,Y 449.852,Z 857.09,A -85,B 0,C 180,E1 7828.079,E2 7828.079} C_VEL
LIN {X 0,Y 449.903,Z 857.089,A -85,B 0,C 180,E1 7831.924,E2 7831.924} C_VEL
LIN {X 0,Y 449.949,Z 852.752,A -85,B 0,C 180,E1 7836.742,E2 7836.742} C_VEL
LIN {X 0,Y 450.34,Z 843.303,A -85,B 0,C 180,E1 7841.6,E2 7841.6} C_VEL
LIN {X 0,Y 451.564,Z 828.286,A -85,B 0,C 180,E1 7846.503,E2 7846.503} C_VEL
LIN {X 0,Y 453.825,Z 806.831,A -85,B 0,C 180,E1 7851.395,E2 7851.395} C_VEL
LIN {X 0,Y 457.026,Z 780.516,A -85,B 0,C 180,E1 7855.667,E2 7855.667} C_VEL
LIN {X 0,Y 460.947,Z 750.072,A -85,B 0,C 180,E1 7859.412,E2 7859.412} C_VEL
LIN {X 0,Y 465.174,Z 716.184,A -85,B 0,C 180,E1 7862.547,E2 7862.547} C_VEL
LIN {X 0,Y 469.337,Z 678.92,A -85,B 0,C 180,E1 7865.051,E2 7865.051} C_VEL
LIN {X 0,Y 472.67,Z 640.027,A -85,B 0,C 180,E1 7866.828,E2 7866.828} C_VEL
LIN {X 0,Y 474.431,Z 602.268,A -85,B 0,C 180,E1 7867.88,E2 7867.88} C_VEL
LIN {X 0,Y 450.421,Z 554.379,A -85,B 0,C 180,E1 7871.032,E2 7871.032} C_VEL
LIN {X 0,Y 448.79,Z 549.53,A -85,B 0,C 180,E1 7871.35,E2 7871.35} C_VEL
LIN {X 0,Y 448.756,Z 549.53,A -85,B 0,C 180,E1 7877.728,E2 7877.728} C_VEL
LIN {X 0,Y 448.714,Z 549.53,A -85,B 0,C 180,E1 7883.817,E2 7883.817} C_VEL
LIN {X 0,Y 448.736,Z 549.53,A -85,B 0,C 180,E1 7889.696,E2 7889.696} C_VEL
LIN {X 0,Y 448.921,Z 549.53,A -85,B 0,C 180,E1 7896.199,E2 7896.199} C_VEL
LIN {X 0,Y 449.146,Z 549.53,A -85,B 0,C 180,E1 7902.387,E2 7902.387} C_VEL
LIN {X 0,Y 449.196,Z 549.53,A -85,B 0,C 180,E1 7908.358,E2 7908.358} C_VEL
LIN {X 0,Y 449.561,Z 549.53,A -85,B 0,C 180,E1 7914.206,E2 7914.206} C_VEL
LIN {X 0,Y 449.723,Z 549.53,A -85,B 0,C 180,E1 7919.984,E2 7919.984} C_VEL
LIN {X 0,Y 449.533,Z 549.53,A -85,B 0,C 180,E1 7925.762,E2 7925.762} C_VEL
LIN {X 0,Y 449.347,Z 549.53,A -85,B 0,C 180,E1 7931.605,E2 7931.605} C_VEL
LIN {X 0,Y 449.163,Z 549.53,A -85,B 0,C 180,E1 7937.579,E2 7937.579} C_VEL
LIN {X 0,Y 448.98,Z 549.53,A -85,B 0,C 180,E1 7943.762,E2 7943.762} C_VEL
LIN {X 0,Y 448.88,Z 549.53,A -85,B 0,C 180,E1 7950.256,E2 7950.256} C_VEL
LIN {X 0,Y 448.846,Z 549.53,A -85,B 0,C 180,E1 7957.21,E2 7957.21} C_VEL
LIN {X 0,Y 448.712,Z 549.53,A -85,B 0,C 180,E1 7962.279,E2 7962.279} C_VEL
LIN {X 0,Y 448.694,Z 549.53,A -85,B 0,C 180,E1 7967.728,E2 7967.728} C_VEL
LIN {X 0,Y 448.86,Z 549.53,A -85,B 0,C 180,E1 7973.744,E2 7973.744} C_VEL
LIN {X 0,Y 448.864,Z 549.53,A -85,B 0,C 180,E1 7979.715,E2 7979.715} C_VEL
LIN {X 0,Y 448.949,Z 549.53,A -85,B 0,C 180,E1 7986.211,E2 7986.211} C_VEL
LIN {X 0,Y 449.128,Z 549.53,A -85,B 0,C 180,E1 7992.397,E2 7992.397} C_VEL
LIN {X 0,Y 449.302,Z 549.53,A -85,B 0,C 180,E1 7998.373,E2 7998.373} C_VEL
LIN {X 0,Y 449.439,Z 549.53,A -85,B 0,C 180,E1 8000.632,E2 8000.632} C_VEL
LIN {X 0,Y 459.861,Z 572.575,A -85,B 0,C 180,E1 8002.168,E2 8002.168} C_VEL
LIN {X 0,Y 469.106,Z 596.676,A -85,B 0,C 180,E1 8003.86,E2 8003.86} C_VEL
LIN {X 0,Y 466.15,Z 632.057,A -85,B 0,C 180,E1 8005.589,E2 8005.589} C_VEL
LIN {X 0,Y 462.315,Z 666.619,A -85,B 0,C 180,E1 8008.128,E2 8008.128} C_VEL
LIN {X 0,Y 458.6,Z 696.256,A -85,B 0,C 180,E1 8011.177,E2 8011.177} C_VEL
LIN {X 0,Y 455.094,Z 723.312,A -85,B 0,C 180,E1 8014.973,E2 8014.973} C_VEL
LIN {X 0,Y 452.54,Z 744.651,A -85,B 0,C 180,E1 8019.112,E2 8019.112} C_VEL
LIN {X 0,Y 450.884,Z 760.932,A -85,B 0,C 180,E1 8023.547,E2 8023.547} C_VEL
LIN {X 0,Y 450.269,Z 770.853,A -85,B 0,C 180,E1 8027.554,E2 8027.554} C_VEL
LIN {X 0,Y 449.727,Z 776.948,A -85,B 0,C 180,E1 8031.658,E2 8031.658} C_VEL
LIN {X 0,Y 449.424,Z 779.107,A -85,B 0,C 180,E1 8035.879,E2 8035.879} C_VEL
LIN {X 0,Y 449.783,Z 777.025,A -85,B 0,C 180,E1 8040.213,E2 8040.213} C_VEL
LIN {X 0,Y 450.375,Z 770.273,A -85,B 0,C 180,E1 8044.72,E2 8044.72} C_VEL
LIN {X 0,Y 451.292,Z 757.744,A -85,B 0,C 180,E1 8049.441,E2 8049.441} C_VEL
LIN {X 0,Y 453.115,Z 739.782,A -85,B 0,C 180,E1 8053.945,E2 8053.945} C_VEL
LIN {X 0,Y 456.014,Z 717.305,A -85,B 0,C 180,E1 8057.974,E2 8057.974} C_VEL
LIN {X 0,Y 459.716,Z 689.565,A -85,B 0,C 180,E1 8061.597,E2 8061.597} C_VEL
LIN {X 0,Y 463.513,Z 659.386,A -85,B 0,C 180,E1 8064.476,E2 8064.476} C_VEL
LIN {X 0,Y 467.129,Z 625.516,A -85,B 0,C 180,E1 8066.781,E2 8066.781} C_VEL
LIN {X 0,Y 468.818,Z 594.91,A -85,B 0,C 180,E1 8068.267,E2 8068.267} C_VEL
LIN {X 0,Y 453.739,Z 560.306,A -85,B 0,C 180,E1 8070.805,E2 8070.805} C_VEL
LIN {X 0,Y 448.918,Z 549.53,A -85,B 0,C 180,E1 8071.601,E2 8071.601} C_VEL
LIN {X 0,Y 449.059,Z 549.53,A -85,B 0,C 180,E1 8078.329,E2 8078.329} C_VEL
LIN {X 0,Y 449.113,Z 549.53,A -85,B 0,C 180,E1 8084.428,E2 8084.428} C_VEL
LIN {X 0,Y 449.313,Z 549.53,A -85,B 0,C 180,E1 8090.351,E2 8090.351} C_VEL
LIN {X 0,Y 449.58,Z 549.53,A -85,B 0,C 180,E1 8096.168,E2 8096.168} C_VEL
LIN {X 0,Y 449.62,Z 549.53,A -85,B 0,C 180,E1 8101.939,E2 8101.939} C_VEL
LIN {X 0,Y 449.468,Z 549.53,A -85,B 0,C 180,E1 8107.732,E2 8107.732} C_VEL
LIN {X 0,Y 449.367,Z 549.53,A -85,B 0,C 180,E1 8113.609,E2 8113.609} C_VEL
LIN {X 0,Y 449.1,Z 549.53,A -85,B 0,C 180,E1 8119.814,E2 8119.814} C_VEL
LIN {X 0,Y 448.939,Z 549.53,A -85,B 0,C 180,E1 8125.922,E2 8125.922} C_VEL
LIN {X 0,Y 448.842,Z 549.53,A -85,B 0,C 180,E1 8132.809,E2 8132.809} C_VEL
LIN {X 0,Y 448.776,Z 549.53,A -85,B 0,C 180,E1 8139.344,E2 8139.344} C_VEL
LIN {X 0,Y 448.619,Z 549.53,A -85,B 0,C 180,E1 8145.061,E2 8145.061} C_VEL
LIN {X 0,Y 448.757,Z 549.53,A -85,B 0,C 180,E1 8148.758,E2 8148.758} C_VEL
LIN {X 0,Y 455.783,Z 564.228,A -85,B 0,C 180,E1 8149.781,E2 8149.781} C_VEL
LIN {X 0,Y 474.518,Z 602.73,A -85,B 0,C 180,E1 8152.205,E2 8152.205} C_VEL
LIN {X 0,Y 472.262,Z 643.467,A -85,B 0,C 180,E1 8153.35,E2 8153.35} C_VEL
LIN {X 0,Y 468.926,Z 681.846,A -85,B 0,C 180,E1 8155.166,E2 8155.166} C_VEL
LIN {X 0,Y 466.683,Z 701.928,A -85,B 0,C 180,E1 8156.438,E2 8156.438} C_VEL
LIN {X 0,Y 461.37,Z 717.074,A -85,B 0,C 180,E1 8157.326,E2 8157.326} C_VEL
LIN {X 0,Y 455.996,Z 731.561,A -85,B 0,C 180,E1 8158.356,E2 8158.356} C_VEL
LIN {X 0,Y 451.63,Z 764.108,A -85,B 0,C 180,E1 8161.841,E2 8161.841} C_VEL
LIN {X 0,Y 447.749,Z 793.038,A -85,B 0,C 180,E1 8165.95,E2 8165.95} C_VEL
LIN {X 0,Y 444.994,Z 816.823,A -85,B 0,C 180,E1 8170.437,E2 8170.437} C_VEL
LIN {X 0,Y 443.299,Z 833.455,A -85,B 0,C 180,E1 8174.705,E2 8174.705} C_VEL
LIN {X 0,Y 442.381,Z 846.721,A -85,B 0,C 180,E1 8179.685,E2 8179.685} C_VEL
LIN {X 0,Y 441.976,Z 853.956,A -85,B 0,C 180,E1 8184.123,E2 8184.123} C_VEL
LIN {X 0,Y 441.947,Z 857.09,A -85,B 0,C 180,E1 8188.045,E2 8188.045} C_VEL
LIN {X 0,Y 441.996,Z 857.09,A -85,B 0,C 180,E1 8191.958,E2 8191.958} C_VEL
LIN {X 0,Y 442.077,Z 852.751,A -85,B 0,C 180,E1 8196.863,E2 8196.863} C_VEL
LIN {X 0,Y 442.489,Z 843.303,A -85,B 0,C 180,E1 8201.809,E2 8201.809} C_VEL
LIN {X 0,Y 443.84,Z 828.285,A -85,B 0,C 180,E1 8206.799,E2 8206.799} C_VEL
LIN {X 0,Y 446.11,Z 806.913,A -85,B 0,C 180,E1 8211.621,E2 8211.621} C_VEL
LIN {X 0,Y 449.556,Z 779.834,A -85,B 0,C 180,E1 8216.106,E2 8216.106} C_VEL
LIN {X 0,Y 453.741,Z 749.196,A -85,B 0,C 180,E1 8219.926,E2 8219.926} C_VEL
LIN {X 0,Y 458.35,Z 714.838,A -85,B 0,C 180,E1 8223.127,E2 8223.127} C_VEL
LIN {X 0,Y 462.621,Z 678.192,A -85,B 0,C 180,E1 8225.61,E2 8225.61} C_VEL
LIN {X 0,Y 466.182,Z 639.165,A -85,B 0,C 180,E1 8227.401,E2 8227.401} C_VEL
LIN {X 0,Y 467.885,Z 604.792,A -85,B 0,C 180,E1 8228.394,E2 8228.394} C_VEL
LIN {X 0,Y 444.741,Z 558.55,A -85,B 0,C 180,E1 8231.523,E2 8231.523} C_VEL
LIN {X 0,Y 440.827,Z 549.53,A -85,B 0,C 180,E1 8232.233,E2 8232.233} C_VEL
LIN {X 0,Y 440.761,Z 549.53,A -85,B 0,C 180,E1 8239.411,E2 8239.411} C_VEL
LIN {X 0,Y 440.794,Z 549.53,A -85,B 0,C 180,E1 8245.249,E2 8245.249} C_VEL
LIN {X 0,Y 440.845,Z 549.53,A -85,B 0,C 180,E1 8251.354,E2 8251.354} C_VEL
LIN {X 0,Y 441.069,Z 549.53,A -85,B 0,C 180,E1 8257.881,E2 8257.881} C_VEL
LIN {X 0,Y 441.175,Z 549.53,A -85,B 0,C 180,E1 8264.106,E2 8264.106} C_VEL
LIN {X 0,Y 441.401,Z 549.53,A -85,B 0,C 180,E1 8270.144,E2 8270.144} C_VEL
LIN {X 0,Y 441.685,Z 549.53,A -85,B 0,C 180,E1 8276.067,E2 8276.067} C_VEL
LIN {X 0,Y 441.751,Z 549.53,A -85,B 0,C 180,E1 8281.941,E2 8281.941} C_VEL
LIN {X 0,Y 441.545,Z 549.53,A -85,B 0,C 180,E1 8287.839,E2 8287.839} C_VEL
LIN {X 0,Y 441.415,Z 549.53,A -85,B 0,C 180,E1 8293.825,E2 8293.825} C_VEL
LIN {X 0,Y 441.171,Z 549.53,A -85,B 0,C 180,E1 8299.979,E2 8299.979} C_VEL
LIN {X 0,Y 440.98,Z 549.53,A -85,B 0,C 180,E1 8306.389,E2 8306.389} C_VEL
LIN {X 0,Y 440.917,Z 549.53,A -85,B 0,C 180,E1 8313.174,E2 8313.174} C_VEL
LIN {X 0,Y 440.866,Z 549.53,A -85,B 0,C 180,E1 8318.068,E2 8318.068} C_VEL
LIN {X 0,Y 440.68,Z 549.53,A -85,B 0,C 180,E1 8324.018,E2 8324.018} C_VEL
LIN {X 0,Y 440.766,Z 549.53,A -85,B 0,C 180,E1 8329.42,E2 8329.42} C_VEL
LIN {X 0,Y 440.979,Z 549.53,A -85,B 0,C 180,E1 8335.164,E2 8335.164} C_VEL
LIN {X 0,Y 440.94,Z 549.53,A -85,B 0,C 180,E1 8341.371,E2 8341.371} C_VEL
LIN {X 0,Y 441.08,Z 549.53,A -85,B 0,C 180,E1 8347.892,E2 8347.892} C_VEL
LIN {X 0,Y 441.293,Z 549.53,A -85,B 0,C 180,E1 8354.122,E2 8354.122} C_VEL
LIN {X 0,Y 441.444,Z 549.53,A -85,B 0,C 180,E1 8359.847,E2 8359.847} C_VEL
LIN {X 0,Y 451.849,Z 571.953,A -85,B 0,C 180,E1 8361.418,E2 8361.418} C_VEL
LIN {X 0,Y 462.421,Z 598.868,A -85,B 0,C 180,E1 8363.389,E2 8363.389} C_VEL
LIN {X 0,Y 459.252,Z 634.083,A -85,B 0,C 180,E1 8365.169,E2 8365.169} C_VEL
LIN {X 0,Y 455.227,Z 668.218,A -85,B 0,C 180,E1 8367.743,E2 8367.743} C_VEL
LIN {X 0,Y 451.144,Z 698.646,A -85,B 0,C 180,E1 8370.957,E2 8370.957} C_VEL
LIN {X 0,Y 447.5,Z 725.086,A -85,B 0,C 180,E1 8374.797,E2 8374.797} C_VEL
LIN {X 0,Y 444.804,Z 746.228,A -85,B 0,C 180,E1 8379.026,E2 8379.026} C_VEL
LIN {X 0,Y 443.154,Z 761.497,A -85,B 0,C 180,E1 8383.287,E2 8383.287} C_VEL
LIN {X 0,Y 442.365,Z 772.437,A -85,B 0,C 180,E1 8387.878,E2 8387.878} C_VEL
LIN {X 0,Y 441.68,Z 778.676,A -85,B 0,C 180,E1 8392.786,E2 8392.786} C_VEL
LIN {X 0,Y 441.58,Z 779.602,A -85,B 0,C 180,E1 8397.376,E2 8397.376} C_VEL
LIN {X 0,Y 442.204,Z 775.467,A -85,B 0,C 180,E1 8402.231,E2 8402.231} C_VEL
LIN {X 0,Y 442.788,Z 766.82,A -85,B 0,C 180,E1 8406.751,E2 8406.751} C_VEL
LIN {X 0,Y 444.148,Z 752.775,A -85,B 0,C 180,E1 8411.328,E2 8411.328} C_VEL
LIN {X 0,Y 446.429,Z 734.003,A -85,B 0,C 180,E1 8415.593,E2 8415.593} C_VEL
LIN {X 0,Y 449.91,Z 709.446,A -85,B 0,C 180,E1 8419.637,E2 8419.637} C_VEL
LIN {X 0,Y 454.052,Z 679.969,A -85,B 0,C 180,E1 8423.147,E2 8423.147} C_VEL
LIN {X 0,Y 458.006,Z 649.145,A -85,B 0,C 180,E1 8425.816,E2 8425.816} C_VEL
LIN {X 0,Y 461.576,Z 614.999,A -85,B 0,C 180,E1 8427.895,E2 8427.895} C_VEL
LIN {X 0,Y 462.19,Z 597.569,A -85,B 0,C 180,E1 8428.734,E2 8428.734} C_VEL
LIN {X 0,Y 447.867,Z 564.24,A -85,B 0,C 180,E1 8431.293,E2 8431.293} C_VEL
LIN {X 0,Y 441.031,Z 550.719,A -85,B 0,C 180,E1 8432.319,E2 8432.319} C_VEL
LIN {X 0,Y 440.953,Z 549.53,A -85,B 0,C 180,E1 8432.361,E2 8432.361} C_VEL
LIN {X 0,Y 441.091,Z 549.53,A -85,B 0,C 180,E1 8437.917,E2 8437.917} C_VEL
LIN {X 0,Y 441.185,Z 549.53,A -85,B 0,C 180,E1 8444.14,E2 8444.14} C_VEL
LIN {X 0,Y 441.408,Z 549.53,A -85,B 0,C 180,E1 8450.177,E2 8450.177} C_VEL
LIN {X 0,Y 441.671,Z 549.53,A -85,B 0,C 180,E1 8456.099,E2 8456.099} C_VEL
LIN {X 0,Y 441.716,Z 549.53,A -85,B 0,C 180,E1 8461.974,E2 8461.974} C_VEL
LIN {X 0,Y 441.555,Z 549.53,A -85,B 0,C 180,E1 8467.872,E2 8467.872} C_VEL
LIN {X 0,Y 441.425,Z 549.53,A -85,B 0,C 180,E1 8473.858,E2 8473.858} C_VEL
LIN {X 0,Y 441.189,Z 549.53,A -85,B 0,C 180,E1 8480.013,E2 8480.013} C_VEL
LIN {X 0,Y 440.969,Z 549.53,A -85,B 0,C 180,E1 8486.426,E2 8486.426} C_VEL
LIN {X 0,Y 440.915,Z 549.53,A -85,B 0,C 180,E1 8493.213,E2 8493.213} C_VEL
LIN {X 0,Y 440.853,Z 549.53,A -85,B 0,C 180,E1 8498.071,E2 8498.071} C_VEL
LIN {X 0,Y 440.636,Z 549.53,A -85,B 0,C 180,E1 8504.016,E2 8504.016} C_VEL
LIN {X 0,Y 440.808,Z 549.721,A -85,B 0,C 180,E1 8507.972,E2 8507.972} C_VEL
LIN {X 0,Y 447.927,Z 564.291,A -85,B 0,C 180,E1 8509.007,E2 8509.007} C_VEL
LIN {X 0,Y 467.767,Z 604.533,A -85,B 0,C 180,E1 8511.669,E2 8511.669} C_VEL
LIN {X 0,Y 465.364,Z 646.903,A -85,B 0,C 180,E1 8512.946,E2 8512.946} C_VEL
LIN {X 0,Y 461.485,Z 687.059,A -85,B 0,C 180,E1 8514.975,E2 8514.975} C_VEL
LIN {X 0,Y 457.143,Z 723.105,A -85,B 0,C 180,E1 8517.614,E2 8517.614} C_VEL
LIN {X 0,Y 455.996,Z 731.561,A -85,B 0,C 180,E1 8518.356,E2 8518.356} C_VEL
LIN {X 0,Y 450.442,Z 745.572,A -85,B 0,C 180,E1 8519.526,E2 8519.526} C_VEL
LIN {X 0,Y 444.967,Z 758.744,A -85,B 0,C 180,E1 8520.8,E2 8520.8} C_VEL
LIN {X 0,Y 440.72,Z 788.671,A -85,B 0,C 180,E1 8524.938,E2 8524.938} C_VEL
LIN {X 0,Y 437.359,Z 814.852,A -85,B 0,C 180,E1 8529.818,E2 8529.818} C_VEL
LIN {X 0,Y 435.347,Z 834.668,A -85,B 0,C 180,E1 8534.933,E2 8534.933} C_VEL
LIN {X 0,Y 434.509,Z 846.721,A -85,B 0,C 180,E1 8539.496,E2 8539.496} C_VEL
LIN {X 0,Y 434.082,Z 853.955,A -85,B 0,C 180,E1 8544.015,E2 8544.015} C_VEL
LIN {X 0,Y 434.041,Z 857.09,A -85,B 0,C 180,E1 8548.009,E2 8548.009} C_VEL
LIN {X 0,Y 434.089,Z 857.089,A -85,B 0,C 180,E1 8551.994,E2 8551.994} C_VEL
LIN {X 0,Y 434.198,Z 852.751,A -85,B 0,C 180,E1 8556.988,E2 8556.988} C_VEL
LIN {X 0,Y 434.759,Z 842.25,A -85,B 0,C 180,E1 8562.457,E2 8562.457} C_VEL
LIN {X 0,Y 436.246,Z 825.693,A -85,B 0,C 180,E1 8567.62,E2 8567.62} C_VEL
LIN {X 0,Y 438.748,Z 803.584,A -85,B 0,C 180,E1 8572.498,E2 8572.498} C_VEL
LIN {X 0,Y 442.406,Z 776.907,A -85,B 0,C 180,E1 8576.879,E2 8576.879} C_VEL
LIN {X 0,Y 446.822,Z 746.896,A -85,B 0,C 180,E1 8580.608,E2 8580.608} C_VEL
LIN {X 0,Y 451.532,Z 713.51,A -85,B 0,C 180,E1 8583.726,E2 8583.726} C_VEL
LIN {X 0,Y 455.981,Z 677.535,A -85,B 0,C 180,E1 8586.178,E2 8586.178} C_VEL
LIN {X 0,Y 459.712,Z 638.58,A -85,B 0,C 180,E1 8587.978,E2 8587.978} C_VEL
LIN {X 0,Y 461.258,Z 607.186,A -85,B 0,C 180,E1 8588.931,E2 8588.931} C_VEL
LIN {X 0,Y 438.013,Z 560.307,A -85,B 0,C 180,E1 8592.191,E2 8592.191} C_VEL
LIN {X 0,Y 432.933,Z 550.745,A -85,B 0,C 180,E1 8592.939,E2 8592.939} C_VEL
LIN {X 0,Y 432.818,Z 549.53,A -85,B 0,C 180,E1 8593.192,E2 8593.192} C_VEL
LIN {X 0,Y 432.831,Z 549.53,A -85,B 0,C 180,E1 8598.506,E2 8598.506} C_VEL
LIN {X 0,Y 432.821,Z 549.53,A -85,B 0,C 180,E1 8603.641,E2 8603.641} C_VEL
LIN {X 0,Y 432.797,Z 549.53,A -85,B 0,C 180,E1 8608.455,E2 8608.455} C_VEL
LIN {X 0,Y 433.018,Z 549.53,A -85,B 0,C 180,E1 8615.268,E2 8615.268} C_VEL
LIN {X 0,Y 433.283,Z 549.53,A -85,B 0,C 180,E1 8621.72,E2 8621.72} C_VEL
LIN {X 0,Y 433.331,Z 549.53,A -85,B 0,C 180,E1 8627.926,E2 8627.926} C_VEL
LIN {X 0,Y 433.739,Z 549.53,A -85,B 0,C 180,E1 8633.994,E2 8633.994} C_VEL
LIN {X 0,Y 433.921,Z 549.53,A -85,B 0,C 180,E1 8639.983,E2 8639.983} C_VEL
LIN {X 0,Y 433.713,Z 549.53,A -85,B 0,C 180,E1 8645.973,E2 8645.973} C_VEL
LIN {X 0,Y 433.484,Z 549.53,A -85,B 0,C 180,E1 8652.905,E2 8652.905} C_VEL
LIN {X 0,Y 433.284,Z 549.53,A -85,B 0,C 180,E1 8658.245,E2 8658.245} C_VEL
LIN {X 0,Y 433.081,Z 549.53,A -85,B 0,C 180,E1 8665.047,E2 8665.047} C_VEL
LIN {X 0,Y 432.978,Z 549.53,A -85,B 0,C 180,E1 8671.491,E2 8671.491} C_VEL
LIN {X 0,Y 432.926,Z 549.53,A -85,B 0,C 180,E1 8676.706,E2 8676.706} C_VEL
LIN {X 0,Y 432.811,Z 549.53,A -85,B 0,C 180,E1 8682.929,E2 8682.929} C_VEL
LIN {X 0,Y 432.809,Z 549.53,A -85,B 0,C 180,E1 8688.511,E2 8688.511} C_VEL
LIN {X 0,Y 432.928,Z 549.53,A -85,B 0,C 180,E1 8693.66,E2 8693.66} C_VEL
LIN {X 0,Y 432.964,Z 549.53,A -85,B 0,C 180,E1 8698.478,E2 8698.478} C_VEL
LIN {X 0,Y 433.066,Z 549.53,A -85,B 0,C 180,E1 8705.281,E2 8705.281} C_VEL
LIN {X 0,Y 433.241,Z 549.53,A -85,B 0,C 180,E1 8711.73,E2 8711.73} C_VEL
LIN {X 0,Y 433.474,Z 549.53,A -85,B 0,C 180,E1 8717.942,E2 8717.942} C_VEL
LIN {X 0,Y 433.473,Z 549.53,A -85,B 0,C 180,E1 8719.023,E2 8719.023} C_VEL
LIN {X 0,Y 440.354,Z 564.17,A -85,B 0,C 180,E1 8720.09,E2 8720.09} C_VEL
LIN {X 0,Y 455.21,Z 599.042,A -85,B 0,C 180,E1 8722.767,E2 8722.767} C_VEL
LIN {X 0,Y 453.493,Z 624.77,A -85,B 0,C 180,E1 8724.053,E2 8724.053} C_VEL
LIN {X 0,Y 449.587,Z 658.833,A -85,B 0,C 180,E1 8726.39,E2 8726.39} C_VEL
LIN {X 0,Y 445.504,Z 689.084,A -85,B 0,C 180,E1 8729.309,E2 8729.309} C_VEL
LIN {X 0,Y 441.347,Z 716.736,A -85,B 0,C 180,E1 8732.938,E2 8732.938} C_VEL
LIN {X 0,Y 438.011,Z 740.096,A -85,B 0,C 180,E1 8737.173,E2 8737.173} C_VEL
LIN {X 0,Y 435.954,Z 757.238,A -85,B 0,C 180,E1 8741.479,E2 8741.479} C_VEL
LIN {X 0,Y 434.794,Z 769.936,A -85,B 0,C 180,E1 8746.119,E2 8746.119} C_VEL
LIN {X 0,Y 434.17,Z 777.042,A -85,B 0,C 180,E1 8750.337,E2 8750.337} C_VEL
LIN {X 0,Y 433.611,Z 780.425,A -85,B 0,C 180,E1 8755.268,E2 8755.268} C_VEL
LIN {X 0,Y 433.931,Z 779.037,A -85,B 0,C 180,E1 8759.67,E2 8759.67} C_VEL
LIN {X 0,Y 434.606,Z 774.08,A -85,B 0,C 180,E1 8763.746,E2 8763.746} C_VEL
LIN {X 0,Y 435.467,Z 763.242,A -85,B 0,C 180,E1 8768.589,E2 8768.589} C_VEL
LIN {X 0,Y 437.339,Z 746.727,A -85,B 0,C 180,E1 8773.351,E2 8773.351} C_VEL
LIN {X 0,Y 440.313,Z 725.784,A -85,B 0,C 180,E1 8777.609,E2 8777.609} C_VEL
LIN {X 0,Y 444.411,Z 698.812,A -85,B 0,C 180,E1 8781.568,E2 8781.568} C_VEL
LIN {X 0,Y 448.745,Z 668.601,A -85,B 0,C 180,E1 8784.799,E2 8784.799} C_VEL
LIN {X 0,Y 453.12,Z 633.822,A -85,B 0,C 180,E1 8787.433,E2 8787.433} C_VEL
LIN {X 0,Y 455.654,Z 600.247,A -85,B 0,C 180,E1 8789.21,E2 8789.21} C_VEL
LIN {X 0,Y 441.032,Z 566.163,A -85,B 0,C 180,E1 8791.95,E2 8791.95} C_VEL
LIN {X 0,Y 433.056,Z 549.995,A -85,B 0,C 180,E1 8793.213,E2 8793.213} C_VEL
LIN {X 0,Y 433.326,Z 549.53,A -85,B 0,C 180,E1 8800.089,E2 8800.089} C_VEL
LIN {X 0,Y 433.298,Z 549.53,A -85,B 0,C 180,E1 8807.189,E2 8807.189} C_VEL
LIN {X 0,Y 433.756,Z 549.53,A -85,B 0,C 180,E1 8814.027,E2 8814.027} C_VEL
LIN {X 0,Y 433.936,Z 549.53,A -85,B 0,C 180,E1 8820.017,E2 8820.017} C_VEL
LIN {X 0,Y 433.717,Z 549.53,A -85,B 0,C 180,E1 8826.007,E2 8826.007} C_VEL
LIN {X 0,Y 433.474,Z 549.53,A -85,B 0,C 180,E1 8832.913,E2 8832.913} C_VEL
LIN {X 0,Y 433.295,Z 549.53,A -85,B 0,C 180,E1 8838.28,E2 8838.28} C_VEL
LIN {X 0,Y 433.036,Z 549.53,A -85,B 0,C 180,E1 8845.041,E2 8845.041} C_VEL
LIN {X 0,Y 432.979,Z 549.53,A -85,B 0,C 180,E1 8851.53,E2 8851.53} C_VEL
LIN {X 0,Y 432.915,Z 549.53,A -85,B 0,C 180,E1 8856.709,E2 8856.709} C_VEL
LIN {X 0,Y 432.705,Z 549.53,A -85,B 0,C 180,E1 8862.918,E2 8862.918} C_VEL
LIN {X 0,Y 432.791,Z 549.556,A -85,B 0,C 180,E1 8867.082,E2 8867.082} C_VEL
LIN {X 0,Y 435.101,Z 555.038,A -85,B 0,C 180,E1 8867.457,E2 8867.457} C_VEL
LIN {X 0,Y 456.141,Z 596.448,A -85,B 0,C 180,E1 8870.443,E2 8870.443} C_VEL
LIN {X 0,Y 461.327,Z 609.294,A -85,B 0,C 180,E1 8871.226,E2 8871.226} C_VEL
LIN {X 0,Y 458.573,Z 648.649,A -85,B 0,C 180,E1 8872.475,E2 8872.475} C_VEL
LIN {X 0,Y 454.702,Z 686.902,A -85,B 0,C 180,E1 8874.454,E2 8874.454} C_VEL
LIN {X 0,Y 450.191,Z 721.998,A -85,B 0,C 180,E1 8877.049,E2 8877.049} C_VEL
LIN {X 0,Y 445.387,Z 755.671,A -85,B 0,C 180,E1 8880.438,E2 8880.438} C_VEL
LIN {X 0,Y 444.967,Z 758.744,A -85,B 0,C 180,E1 8880.8,E2 8880.8} C_VEL
LIN {X 0,Y 439.357,Z 771.379,A -85,B 0,C 180,E1 8882.207,E2 8882.207} C_VEL
LIN {X 0,Y 434.145,Z 781.776,A -85,B 0,C 180,E1 8883.534,E2 8883.534} C_VEL
LIN {X 0,Y 433.88,Z 783.171,A -85,B 0,C 180,E1 8883.752,E2 8883.752} C_VEL
LIN {X 0,Y 430.393,Z 808.037,A -85,B 0,C 180,E1 8888.17,E2 8888.17} C_VEL
LIN {X 0,Y 428.08,Z 827.668,A -85,B 0,C 180,E1 8892.815,E2 8892.815} C_VEL
LIN {X 0,Y 426.811,Z 842.692,A -85,B 0,C 180,E1 8897.754,E2 8897.754} C_VEL
LIN {X 0,Y 426.285,Z 851.952,A -85,B 0,C 180,E1 8902.41,E2 8902.41} C_VEL
LIN {X 0,Y 426.135,Z 857.089,A -85,B 0,C 180,E1 8907.972,E2 8907.972} C_VEL
LIN {X 0,Y 426.183,Z 857.089,A -85,B 0,C 180,E1 8912.031,E2 8912.031} C_VEL
LIN {X 0,Y 426.288,Z 851.951,A -85,B 0,C 180,E1 8917.593,E2 8917.593} C_VEL
LIN {X 0,Y 426.896,Z 841.732,A -85,B 0,C 180,E1 8922.643,E2 8922.643} C_VEL
LIN {X 0,Y 428.37,Z 826.26,A -85,B 0,C 180,E1 8927.612,E2 8927.612} C_VEL
LIN {X 0,Y 430.963,Z 804.187,A -85,B 0,C 180,E1 8932.656,E2 8932.656} C_VEL
LIN {X 0,Y 434.839,Z 777.586,A -85,B 0,C 180,E1 8937.155,E2 8937.155} C_VEL
LIN {X 0,Y 439.535,Z 747.453,A -85,B 0,C 180,E1 8940.998,E2 8940.998} C_VEL
LIN {X 0,Y 444.633,Z 713.457,A -85,B 0,C 180,E1 8944.237,E2 8944.237} C_VEL
LIN {X 0,Y 449.379,Z 676.725,A -85,B 0,C 180,E1 8946.771,E2 8946.771} C_VEL
LIN {X 0,Y 453.241,Z 638.474,A -85,B 0,C 180,E1 8948.554,E2 8948.554} C_VEL
LIN {X 0,Y 454.997,Z 610.347,A -85,B 0,C 180,E1 8949.414,E2 8949.414} C_VEL
LIN {X 0,Y 433.137,Z 565.817,A -85,B 0,C 180,E1 8952.6,E2 8952.6} C_VEL
LIN {X 0,Y 424.969,Z 550.578,A -85,B 0,C 180,E1 8953.837,E2 8953.837} C_VEL
LIN {X 0,Y 424.912,Z 549.53,A -85,B 0,C 180,E1 8953.93,E2 8953.93} C_VEL
LIN {X 0,Y 424.892,Z 549.53,A -85,B 0,C 180,E1 8960.252,E2 8960.252} C_VEL
LIN {X 0,Y 424.854,Z 549.53,A -85,B 0,C 180,E1 8965.357,E2 8965.357} C_VEL
LIN {X 0,Y 424.896,Z 549.53,A -85,B 0,C 180,E1 8970.173,E2 8970.173} C_VEL
LIN {X 0,Y 425.21,Z 549.53,A -85,B 0,C 180,E1 8977.329,E2 8977.329} C_VEL
LIN {X 0,Y 425.346,Z 549.53,A -85,B 0,C 180,E1 8983.498,E2 8983.498} C_VEL
LIN {X 0,Y 425.529,Z 549.53,A -85,B 0,C 180,E1 8989.772,E2 8989.772} C_VEL
LIN {X 0,Y 425.868,Z 549.53,A -85,B 0,C 180,E1 8995.92,E2 8995.92} C_VEL
LIN {X 0,Y 425.941,Z 549.53,A -85,B 0,C 180,E1 9002.013,E2 9002.013} C_VEL
LIN {X 0,Y 425.705,Z 549.53,A -85,B 0,C 180,E1 9008.132,E2 9008.132} C_VEL
LIN {X 0,Y 425.533,Z 549.53,A -85,B 0,C 180,E1 9014.352,E2 9014.352} C_VEL
LIN {X 0,Y 425.278,Z 549.53,A -85,B 0,C 180,E1 9020.76,E2 9020.76} C_VEL
LIN {X 0,Y 425.1,Z 549.53,A -85,B 0,C 180,E1 9027.456,E2 9027.456} C_VEL
LIN {X 0,Y 425.075,Z 549.53,A -85,B 0,C 180,E1 9032.146,E2 9032.146} C_VEL
LIN {X 0,Y 424.952,Z 549.53,A -85,B 0,C 180,E1 9038.625,E2 9038.625} C_VEL
LIN {X 0,Y 424.853,Z 549.53,A -85,B 0,C 180,E1 9045.227,E2 9045.227} C_VEL
LIN {X 0,Y 424.935,Z 549.53,A -85,B 0,C 180,E1 9051.332,E2 9051.332} C_VEL
LIN {X 0,Y 425.068,Z 549.53,A -85,B 0,C 180,E1 9058.377,E2 9058.377} C_VEL
LIN {X 0,Y 425.154,Z 549.53,A -85,B 0,C 180,E1 9064.789,E2 9064.789} C_VEL
LIN {X 0,Y 425.317,Z 549.53,A -85,B 0,C 180,E1 9071.377,E2 9071.377} C_VEL
LIN {X 0,Y 425.579,Z 549.53,A -85,B 0,C 180,E1 9078.169,E2 9078.169} C_VEL
LIN {X 0,Y 432.119,Z 563.585,A -85,B 0,C 180,E1 9079.235,E2 9079.235} C_VEL
LIN {X 0,Y 446.378,Z 595.763,A -85,B 0,C 180,E1 9081.811,E2 9081.811} C_VEL
LIN {X 0,Y 448.945,Z 605.278,A -85,B 0,C 180,E1 9082.515,E2 9082.515} C_VEL
LIN {X 0,Y 445.514,Z 637.95,A -85,B 0,C 180,E1 9084.288,E2 9084.288} C_VEL
LIN {X 0,Y 441.126,Z 671.39,A -85,B 0,C 180,E1 9086.935,E2 9086.935} C_VEL
LIN {X 0,Y 436.653,Z 701.366,A -85,B 0,C 180,E1 9090.246,E2 9090.246} C_VEL
LIN {X 0,Y 432.464,Z 727.82,A -85,B 0,C 180,E1 9094.284,E2 9094.284} C_VEL
LIN {X 0,Y 429.536,Z 748.166,A -85,B 0,C 180,E1 9098.549,E2 9098.549} C_VEL
LIN {X 0,Y 427.582,Z 763.772,A -85,B 0,C 180,E1 9103.134,E2 9103.134} C_VEL
LIN {X 0,Y 426.777,Z 773.52,A -85,B 0,C 180,E1 9107.416,E2 9107.416} C_VEL
LIN {X 0,Y 426.235,Z 778.317,A -85,B 0,C 180,E1 9110.733,E2 9110.733} C_VEL
LIN {X 0,Y 425.762,Z 781.113,A -85,B 0,C 180,E1 9115.169,E2 9115.169} C_VEL
LIN {X 0,Y 426.081,Z 779.765,A -85,B 0,C 180,E1 9119.722,E2 9119.722} C_VEL
LIN {X 0,Y 426.837,Z 773.82,A -85,B 0,C 180,E1 9124.446,E2 9124.446} C_VEL
LIN {X 0,Y 427.937,Z 762.347,A -85,B 0,C 180,E1 9129.398,E2 9129.398} C_VEL
LIN {X 0,Y 430.098,Z 745.062,A -85,B 0,C 180,E1 9134.261,E2 9134.261} C_VEL
LIN {X 0,Y 433.523,Z 722.841,A -85,B 0,C 180,E1 9138.631,E2 9138.631} C_VEL
LIN {X 0,Y 437.834,Z 696.308,A -85,B 0,C 180,E1 9142.436,E2 9142.436} C_VEL
LIN {X 0,Y 442.65,Z 664.337,A -85,B 0,C 180,E1 9145.757,E2 9145.757} C_VEL
LIN {X 0,Y 446.99,Z 630.578,A -85,B 0,C 180,E1 9148.219,E2 9148.219} C_VEL
LIN {X 0,Y 449.588,Z 604.411,A -85,B 0,C 180,E1 9149.576,E2 9149.576} C_VEL
LIN {X 0,Y 435.261,Z 569.913,A -85,B 0,C 180,E1 9152.47,E2 9152.47} C_VEL
LIN {X 0,Y 425.173,Z 550.183,A -85,B 0,C 180,E1 9154.125,E2 9154.125} C_VEL
LIN {X 0,Y 425.305,Z 549.53,A -85,B 0,C 180,E1 9159.242,E2 9159.242} C_VEL
LIN {X 0,Y 425.371,Z 549.53,A -85,B 0,C 180,E1 9165.642,E2 9165.642} C_VEL
LIN {X 0,Y 425.701,Z 549.53,A -85,B 0,C 180,E1 9171.868,E2 9171.868} C_VEL
LIN {X 0,Y 426.074,Z 549.53,A -85,B 0,C 180,E1 9177.988,E2 9177.988} C_VEL
LIN {X 0,Y 425.913,Z 549.53,A -85,B 0,C 180,E1 9184.079,E2 9184.079} C_VEL
LIN {X 0,Y 425.664,Z 549.53,A -85,B 0,C 180,E1 9190.225,E2 9190.225} C_VEL
LIN {X 0,Y 425.417,Z 549.53,A -85,B 0,C 180,E1 9196.724,E2 9196.724} C_VEL
LIN {X 0,Y 425.217,Z 549.53,A -85,B 0,C 180,E1 9202.99,E2 9202.99} C_VEL
LIN {X 0,Y 425.049,Z 549.53,A -85,B 0,C 180,E1 9209.815,E2 9209.815} C_VEL
LIN {X 0,Y 424.977,Z 549.53,A -85,B 0,C 180,E1 9217.142,E2 9217.142} C_VEL
LIN {X 0,Y 424.81,Z 549.53,A -85,B 0,C 180,E1 9222.458,E2 9222.458} C_VEL
LIN {X 0,Y 424.871,Z 550.193,A -85,B 0,C 180,E1 9226.17,E2 9226.17} C_VEL
LIN {X 0,Y 448.798,Z 596.858,A -85,B 0,C 180,E1 9229.751,E2 9229.751} C_VEL
LIN {X 0,Y 454.804,Z 611.807,A -85,B 0,C 180,E1 9230.707,E2 9230.707} C_VEL
LIN {X 0,Y 451.855,Z 650.256,A -85,B 0,C 180,E1 9231.983,E2 9231.983} C_VEL
LIN {X 0,Y 447.804,Z 687.776,A -85,B 0,C 180,E1 9233.983,E2 9233.983} C_VEL
LIN {X 0,Y 443.125,Z 722.235,A -85,B 0,C 180,E1 9236.588,E2 9236.588} C_VEL
LIN {X 0,Y 438.215,Z 754.736,A -85,B 0,C 180,E1 9239.91,E2 9239.91} C_VEL
LIN {X 0,Y 433.88,Z 783.171,A -85,B 0,C 180,E1 9243.752,E2 9243.752} C_VEL
LIN {X 0,Y 430.386,Z 791.612,A -85,B 0,C 180,E1 9245.017,E2 9245.017} C_VEL
LIN {X 0,Y 423.458,Z 803.247,A -85,B 0,C 180,E1 9246.954,E2 9246.954} C_VEL
LIN {X 0,Y 423.162,Z 804.497,A -85,B 0,C 180,E1 9247.194,E2 9247.194} C_VEL
LIN {X 0,Y 420.423,Z 825.839,A -85,B 0,C 180,E1 9252.188,E2 9252.188} C_VEL
LIN {X 0,Y 418.935,Z 841.93,A -85,B 0,C 180,E1 9257.52,E2 9257.52} C_VEL
LIN {X 0,Y 418.38,Z 851.643,A -85,B 0,C 180,E1 9262.535,E2 9262.535} C_VEL
LIN {X 0,Y 418.25,Z 856.578,A -85,B 0,C 180,E1 9267.934,E2 9267.934} C_VEL
LIN {X 0,Y 418.294,Z 856.586,A -85,B 0,C 180,E1 9272.069,E2 9272.069} C_VEL
LIN {X 0,Y 418.386,Z 851.668,A -85,B 0,C 180,E1 9277.469,E2 9277.469} C_VEL
LIN {X 0,Y 418.967,Z 841.999,A -85,B 0,C 180,E1 9282.482,E2 9282.482} C_VEL
LIN {X 0,Y 420.547,Z 825.878,A -85,B 0,C 180,E1 9287.85,E2 9287.85} C_VEL
LIN {X 0,Y 423.438,Z 803.419,A -85,B 0,C 180,E1 9293.081,E2 9293.081} C_VEL
LIN {X 0,Y 427.428,Z 777.461,A -85,B 0,C 180,E1 9297.558,E2 9297.558} C_VEL
LIN {X 0,Y 432.481,Z 746.577,A -85,B 0,C 180,E1 9301.561,E2 9301.561} C_VEL
LIN {X 0,Y 437.693,Z 713.877,A -85,B 0,C 180,E1 9304.722,E2 9304.722} C_VEL
LIN {X 0,Y 442.629,Z 677.522,A -85,B 0,C 180,E1 9307.287,E2 9307.287} C_VEL
LIN {X 0,Y 446.701,Z 639.558,A -85,B 0,C 180,E1 9309.102,E2 9309.102} C_VEL
LIN {X 0,Y 448.465,Z 612.928,A -85,B 0,C 180,E1 9309.954,E2 9309.954} C_VEL
LIN {X 0,Y 428.502,Z 571.763,A -85,B 0,C 180,E1 9312.983,E2 9312.983} C_VEL
LIN {X 0,Y 417.084,Z 550.634,A -85,B 0,C 180,E1 9314.764,E2 9314.764} C_VEL
LIN {X 0,Y 417.017,Z 549.53,A -85,B 0,C 180,E1 9315.043,E2 9315.043} C_VEL
LIN {X 0,Y 417.002,Z 549.53,A -85,B 0,C 180,E1 9322.023,E2 9322.023} C_VEL
LIN {X 0,Y 416.959,Z 549.53,A -85,B 0,C 180,E1 9329.545,E2 9329.545} C_VEL
LIN {X 0,Y 417.187,Z 549.53,A -85,B 0,C 180,E1 9336.541,E2 9336.541} C_VEL
LIN {X 0,Y 417.433,Z 549.53,A -85,B 0,C 180,E1 9343.176,E2 9343.176} C_VEL
LIN {X 0,Y 417.592,Z 549.53,A -85,B 0,C 180,E1 9349.576,E2 9349.576} C_VEL
LIN {X 0,Y 417.956,Z 549.53,A -85,B 0,C 180,E1 9355.843,E2 9355.843} C_VEL
LIN {X 0,Y 418.065,Z 549.53,A -85,B 0,C 180,E1 9362.051,E2 9362.051} C_VEL
LIN {X 0,Y 417.783,Z 549.53,A -85,B 0,C 180,E1 9368.288,E2 9368.288} C_VEL
LIN {X 0,Y 417.601,Z 549.53,A -85,B 0,C 180,E1 9374.631,E2 9374.631} C_VEL
LIN {X 0,Y 417.348,Z 549.53,A -85,B 0,C 180,E1 9381.173,E2 9381.173} C_VEL
LIN {X 0,Y 417.12,Z 549.53,A -85,B 0,C 180,E1 9388.027,E2 9388.027} C_VEL
LIN {X 0,Y 417.084,Z 549.53,A -85,B 0,C 180,E1 9395.341,E2 9395.341} C_VEL
LIN {X 0,Y 416.975,Z 549.53,A -85,B 0,C 180,E1 9400.614,E2 9400.614} C_VEL
LIN {X 0,Y 416.876,Z 549.53,A -85,B 0,C 180,E1 9406.545,E2 9406.545} C_VEL
LIN {X 0,Y 417.063,Z 549.53,A -85,B 0,C 180,E1 9412.704,E2 9412.704} C_VEL
LIN {X 0,Y 417.119,Z 549.53,A -85,B 0,C 180,E1 9419.569,E2 9419.569} C_VEL
LIN {X 0,Y 417.251,Z 549.53,A -85,B 0,C 180,E1 9426.556,E2 9426.556} C_VEL
LIN {X 0,Y 417.465,Z 549.53,A -85,B 0,C 180,E1 9433.19,E2 9433.19} C_VEL
LIN {X 0,Y 417.615,Z 549.53,A -85,B 0,C 180,E1 9437.286,E2 9437.286} C_VEL
LIN {X 0,Y 422.568,Z 560.13,A -85,B 0,C 180,E1 9438.12,E2 9438.12} C_VEL
LIN {X 0,Y 438.066,Z 593.655,A -85,B 0,C 180,E1 9440.915,E2 9440.915} C_VEL
LIN {X 0,Y 442.395,Z 606.434,A -85,B 0,C 180,E1 9441.967,E2 9441.967} C_VEL
LIN {X 0,Y 438.743,Z 639.504,A -85,B 0,C 180,E1 9443.804,E2 9443.804} C_VEL
LIN {X 0,Y 434.108,Z 672.963,A -85,B 0,C 180,E1 9446.511,E2 9446.511} C_VEL
LIN {X 0,Y 429.229,Z 703.603,A -85,B 0,C 180,E1 9449.998,E2 9449.998} C_VEL
LIN {X 0,Y 424.92,Z 729.493,A -85,B 0,C 180,E1 9454.071,E2 9454.071} C_VEL
LIN {X 0,Y 421.681,Z 750.559,A -85,B 0,C 180,E1 9458.65,E2 9458.65} C_VEL
LIN {X 0,Y 419.761,Z 765.275,A -85,B 0,C 180,E1 9463.181,E2 9463.181} C_VEL
LIN {X 0,Y 418.877,Z 775.105,A -85,B 0,C 180,E1 9467.755,E2 9467.755} C_VEL
LIN {X 0,Y 418.303,Z 779.583,A -85,B 0,C 180,E1 9471.144,E2 9471.144} C_VEL
LIN {X 0,Y 417.867,Z 781.912,A -85,B 0,C 180,E1 9475.678,E2 9475.678} C_VEL
LIN {X 0,Y 418.305,Z 780.059,A -85,B 0,C 180,E1 9480.332,E2 9480.332} C_VEL
LIN {X 0,Y 419.077,Z 773.561,A -85,B 0,C 180,E1 9485.177,E2 9485.177} C_VEL
LIN {X 0,Y 420.391,Z 761.398,A -85,B 0,C 180,E1 9490.248,E2 9490.248} C_VEL
LIN {X 0,Y 422.932,Z 743.188,A -85,B 0,C 180,E1 9495.205,E2 9495.205} C_VEL
LIN {X 0,Y 426.719,Z 720.814,A -85,B 0,C 180,E1 9499.522,E2 9499.522} C_VEL
LIN {X 0,Y 431.512,Z 693.039,A -85,B 0,C 180,E1 9503.409,E2 9503.409} C_VEL
LIN {X 0,Y 436.313,Z 662.597,A -85,B 0,C 180,E1 9506.499,E2 9506.499} C_VEL
LIN {X 0,Y 440.826,Z 628.298,A -85,B 0,C 180,E1 9508.969,E2 9508.969} C_VEL
LIN {X 0,Y 442.792,Z 606.434,A -85,B 0,C 180,E1 9510.131,E2 9510.131} C_VEL
LIN {X 0,Y 429.433,Z 573.905,A -85,B 0,C 180,E1 9512.985,E2 9512.985} C_VEL
LIN {X 0,Y 417.421,Z 551.25,A -85,B 0,C 180,E1 9515.053,E2 9515.053} C_VEL
LIN {X 0,Y 417.218,Z 549.53,A -85,B 0,C 180,E1 9515.121,E2 9515.121} C_VEL
LIN {X 0,Y 417.415,Z 549.53,A -85,B 0,C 180,E1 9521.035,E2 9521.035} C_VEL
LIN {X 0,Y 417.529,Z 549.53,A -85,B 0,C 180,E1 9527.497,E2 9527.497} C_VEL
LIN {X 0,Y 417.933,Z 549.53,A -85,B 0,C 180,E1 9533.8,E2 9533.8} C_VEL
LIN {X 0,Y 418.141,Z 549.53,A -85,B 0,C 180,E1 9540.017,E2 9540.017} C_VEL
LIN {X 0,Y 417.881,Z 549.53,A -85,B 0,C 180,E1 9546.235,E2 9546.235} C_VEL
LIN {X 0,Y 417.674,Z 549.53,A -85,B 0,C 180,E1 9552.721,E2 9552.721} C_VEL
LIN {X 0,Y 417.412,Z 549.53,A -85,B 0,C 180,E1 9559.001,E2 9559.001} C_VEL
LIN {X 0,Y 417.174,Z 549.53,A -85,B 0,C 180,E1 9565.739,E2 9565.739} C_VEL
LIN {X 0,Y 417.129,Z 549.53,A -85,B 0,C 180,E1 9570.441,E2 9570.441} C_VEL
LIN {X 0,Y 417.083,Z 549.53,A -85,B 0,C 180,E1 9577.256,E2 9577.256} C_VEL
LIN {X 0,Y 416.879,Z 549.53,A -85,B 0,C 180,E1 9584.662,E2 9584.662} C_VEL
LIN {X 0,Y 416.889,Z 549.53,A -85,B 0,C 180,E1 9585.162,E2 9585.162} C_VEL
LIN {X 0,Y 419.37,Z 555.266,A -85,B 0,C 180,E1 9585.608,E2 9585.608} C_VEL
LIN {X 0,Y 440.645,Z 595.447,A -85,B 0,C 180,E1 9588.895,E2 9588.895} C_VEL
LIN {X 0,Y 448.294,Z 614.228,A -85,B 0,C 180,E1 9590.167,E2 9590.167} C_VEL
LIN {X 0,Y 444.964,Z 653.734,A -85,B 0,C 180,E1 9591.555,E2 9591.555} C_VEL
LIN {X 0,Y 440.23,Z 693.774,A -85,B 0,C 180,E1 9593.827,E2 9593.827} C_VEL
LIN {X 0,Y 434.813,Z 730.632,A -85,B 0,C 180,E1 9596.868,E2 9596.868} C_VEL
LIN {X 0,Y 429.554,Z 763.248,A -85,B 0,C 180,E1 9600.542,E2 9600.542} C_VEL
LIN {X 0,Y 425.044,Z 791.522,A -85,B 0,C 180,E1 9604.786,E2 9604.786} C_VEL
LIN {X 0,Y 423.162,Z 804.497,A -85,B 0,C 180,E1 9607.194,E2 9607.194} C_VEL
LIN {X 0,Y 417.956,Z 813.854,A -85,B 0,C 180,E1 9609.089,E2 9609.089} C_VEL
LIN {X 0,Y 413.018,Z 822.283,A -85,B 0,C 180,E1 9611.106,E2 9611.106} C_VEL
LIN {X 0,Y 411.354,Z 838.27,A -85,B 0,C 180,E1 9616.144,E2 9616.144} C_VEL
LIN {X 0,Y 410.734,Z 847.869,A -85,B 0,C 180,E1 9620.485,E2 9620.485} C_VEL
LIN {X 0,Y 410.356,Z 854.6,A -85,B 0,C 180,E1 9625.784,E2 9625.784} C_VEL
LIN {X 0,Y 410.422,Z 856.315,A -85,B 0,C 180,E1 9630.002,E2 9630.002} C_VEL
LIN {X 0,Y 410.374,Z 853.717,A -85,B 0,C 180,E1 9635.276,E2 9635.276} C_VEL
LIN {X 0,Y 410.769,Z 845.906,A -85,B 0,C 180,E1 9640.586,E2 9640.586} C_VEL
LIN {X 0,Y 411.909,Z 832.493,A -85,B 0,C 180,E1 9645.949,E2 9645.949} C_VEL
LIN {X 0,Y 414.335,Z 812.693,A -85,B 0,C 180,E1 9651.36,E2 9651.36} C_VEL
LIN {X 0,Y 418.503,Z 786.509,A -85,B 0,C 180,E1 9656.502,E2 9656.502} C_VEL
LIN {X 0,Y 423.399,Z 757.706,A -85,B 0,C 180,E1 9660.707,E2 9660.707} C_VEL
LIN {X 0,Y 428.935,Z 725.178,A -85,B 0,C 180,E1 9664.258,E2 9664.258} C_VEL
LIN {X 0,Y 434.52,Z 688.982,A -85,B 0,C 180,E1 9667.138,E2 9667.138} C_VEL
LIN {X 0,Y 439.155,Z 651.335,A -85,B 0,C 180,E1 9669.214,E2 9669.214} C_VEL
LIN {X 0,Y 441.894,Z 615.456,A -85,B 0,C 180,E1 9670.514,E2 9670.514} C_VEL
LIN {X 0,Y 424.166,Z 578.208,A -85,B 0,C 180,E1 9673.331,E2 9673.331} C_VEL
LIN {X 0,Y 409.071,Z 550.021,A -85,B 0,C 180,E1 9675.766,E2 9675.766} C_VEL
LIN {X 0,Y 408.996,Z 549.53,A -85,B 0,C 180,E1 9681.143,E2 9681.143} C_VEL
LIN {X 0,Y 408.966,Z 549.53,A -85,B 0,C 180,E1 9688.069,E2 9688.069} C_VEL
LIN {X 0,Y 409.115,Z 549.53,A -85,B 0,C 180,E1 9693.716,E2 9693.716} C_VEL
LIN {X 0,Y 409.468,Z 549.53,A -85,B 0,C 180,E1 9700.616,E2 9700.616} C_VEL
LIN {X 0,Y 409.584,Z 549.53,A -85,B 0,C 180,E1 9707.214,E2 9707.214} C_VEL
LIN {X 0,Y 409.987,Z 549.53,A -85,B 0,C 180,E1 9713.644,E2 9713.644} C_VEL
LIN {X 0,Y 410.229,Z 549.53,A -85,B 0,C 180,E1 9719.982,E2 9719.982} C_VEL
LIN {X 0,Y 409.975,Z 549.53,A -85,B 0,C 180,E1 9726.369,E2 9726.369} C_VEL
LIN {X 0,Y 409.767,Z 549.53,A -85,B 0,C 180,E1 9732.744,E2 9732.744} C_VEL
LIN {X 0,Y 409.47,Z 549.53,A -85,B 0,C 180,E1 9739.347,E2 9739.347} C_VEL
LIN {X 0,Y 409.226,Z 549.53,A -85,B 0,C 180,E1 9746.237,E2 9746.237} C_VEL
LIN {X 0,Y 409.162,Z 549.53,A -85,B 0,C 180,E1 9753.557,E2 9753.557} C_VEL
LIN {X 0,Y 409.002,Z 549.53,A -85,B 0,C 180,E1 9759.211,E2 9759.211} C_VEL
LIN {X 0,Y 408.878,Z 549.53,A -85,B 0,C 180,E1 9765.473,E2 9765.473} C_VEL
LIN {X 0,Y 409.002,Z 549.53,A -85,B 0,C 180,E1 9771.153,E2 9771.153} C_VEL
LIN {X 0,Y 409.154,Z 549.53,A -85,B 0,C 180,E1 9776.41,E2 9776.41} C_VEL
LIN {X 0,Y 409.202,Z 549.53,A -85,B 0,C 180,E1 9783.733,E2 9783.733} C_VEL
LIN {X 0,Y 409.431,Z 549.53,A -85,B 0,C 180,E1 9790.626,E2 9790.626} C_VEL
LIN {X 0,Y 409.636,Z 549.53,A -85,B 0,C 180,E1 9796.348,E2 9796.348} C_VEL
LIN {X 0,Y 414.145,Z 559.314,A -85,B 0,C 180,E1 9797.141,E2 9797.141} C_VEL
LIN {X 0,Y 429.769,Z 592.015,A -85,B 0,C 180,E1 9799.998,E2 9799.998} C_VEL
LIN {X 0,Y 435.692,Z 609.682,A -85,B 0,C 180,E1 9801.503,E2 9801.503} C_VEL
LIN {X 0,Y 431.684,Z 643.541,A -85,B 0,C 180,E1 9803.475,E2 9803.475} C_VEL
LIN {X 0,Y 426.69,Z 677.04,A -85,B 0,C 180,E1 9806.323,E2 9806.323} C_VEL
LIN {X 0,Y 421.688,Z 706.536,A -85,B 0,C 180,E1 9809.843,E2 9809.843} C_VEL
LIN {X 0,Y 417.35,Z 731.346,A -85,B 0,C 180,E1 9813.886,E2 9813.886} C_VEL
LIN {X 0,Y 413.834,Z 752.809,A -85,B 0,C 180,E1 9818.746,E2 9818.746} C_VEL
LIN {X 0,Y 411.866,Z 767.142,A -85,B 0,C 180,E1 9823.409,E2 9823.409} C_VEL
LIN {X 0,Y 410.903,Z 776.883,A -85,B 0,C 180,E1 9828.31,E2 9828.31} C_VEL
LIN {X 0,Y 410.128,Z 781.83,A -85,B 0,C 180,E1 9833.173,E2 9833.173} C_VEL
LIN {X 0,Y 410.167,Z 781.992,A -85,B 0,C 180,E1 9838.571,E2 9838.571} C_VEL
LIN {X 0,Y 411.01,Z 777.385,A -85,B 0,C 180,E1 9843.415,E2 9843.415} C_VEL
LIN {X 0,Y 411.988,Z 767.563,A -85,B 0,C 180,E1 9848.509,E2 9848.509} C_VEL
LIN {X 0,Y 414.312,Z 751.172,A -85,B 0,C 180,E1 9853.788,E2 9853.788} C_VEL
LIN {X 0,Y 417.817,Z 730.631,A -85,B 0,C 180,E1 9858.351,E2 9858.351} C_VEL
LIN {X 0,Y 422.576,Z 704.693,A -85,B 0,C 180,E1 9862.522,E2 9862.522} C_VEL
LIN {X 0,Y 427.781,Z 674.414,A -85,B 0,C 180,E1 9866.036,E2 9866.036} C_VEL
LIN {X 0,Y 432.831,Z 641.088,A -85,B 0,C 180,E1 9868.783,E2 9868.783} C_VEL
LIN {X 0,Y 436.304,Z 609.152,A -85,B 0,C 180,E1 9870.64,E2 9870.64} C_VEL
LIN {X 0,Y 422.798,Z 575.793,A -85,B 0,C 180,E1 9873.69,E2 9873.69} C_VEL
LIN {X 0,Y 409.445,Z 550.82,A -85,B 0,C 180,E1 9876.109,E2 9876.109} C_VEL
LIN {X 0,Y 409.347,Z 549.53,A -85,B 0,C 180,E1 9876.263,E2 9876.263} C_VEL
LIN {X 0,Y 409.518,Z 549.53,A -85,B 0,C 180,E1 9883.342,E2 9883.342} C_VEL
LIN {X 0,Y 409.694,Z 549.53,A -85,B 0,C 180,E1 9889.408,E2 9889.408} C_VEL
LIN {X 0,Y 410.034,Z 549.53,A -85,B 0,C 180,E1 9895.798,E2 9895.798} C_VEL
LIN {X 0,Y 410.127,Z 549.53,A -85,B 0,C 180,E1 9902.126,E2 9902.126} C_VEL
LIN {X 0,Y 409.865,Z 549.53,A -85,B 0,C 180,E1 9908.484,E2 9908.484} C_VEL
LIN {X 0,Y 409.66,Z 549.53,A -85,B 0,C 180,E1 9914.957,E2 9914.957} C_VEL
LIN {X 0,Y 409.388,Z 549.53,A -85,B 0,C 180,E1 9921.643,E2 9921.643} C_VEL
LIN {X 0,Y 409.198,Z 549.53,A -85,B 0,C 180,E1 9928.659,E2 9928.659} C_VEL
LIN {X 0,Y 409.14,Z 549.53,A -85,B 0,C 180,E1 9935.768,E2 9935.768} C_VEL
LIN {X 0,Y 408.846,Z 549.53,A -85,B 0,C 180,E1 9942.426,E2 9942.426} C_VEL
LIN {X 0,Y 408.929,Z 549.537,A -85,B 0,C 180,E1 9944.112,E2 9944.112} C_VEL
LIN {X 0,Y 411.168,Z 555.002,A -85,B 0,C 180,E1 9944.544,E2 9944.544} C_VEL
LIN {X 0,Y 430.839,Z 590.657,A -85,B 0,C 180,E1 9947.73,E2 9947.73} C_VEL
LIN {X 0,Y 441.883,Z 615.646,A -85,B 0,C 180,E1 9949.583,E2 9949.583} C_VEL
LIN {X 0,Y 438.157,Z 656.905,A -85,B 0,C 180,E1 9951.105,E2 9951.105} C_VEL
LIN {X 0,Y 433.015,Z 696.871,A -85,B 0,C 180,E1 9953.498,E2 9953.498} C_VEL
LIN {X 0,Y 427.468,Z 732.336,A -85,B 0,C 180,E1 9956.54,E2 9956.54} C_VEL
LIN {X 0,Y 421.949,Z 764.678,A -85,B 0,C 180,E1 9960.308,E2 9960.308} C_VEL
LIN {X 0,Y 417.231,Z 793.006,A -85,B 0,C 180,E1 9964.725,E2 9964.725} C_VEL
LIN {X 0,Y 413.752,Z 816.924,A -85,B 0,C 180,E1 9969.73,E2 9969.73} C_VEL
LIN {X 0,Y 413.018,Z 822.283,A -85,B 0,C 180,E1 9971.106,E2 9971.106} C_VEL
LIN {X 0,Y 408.227,Z 829.84,A -85,B 0,C 180,E1 9973.21,E2 9973.21} C_VEL
LIN {X 0,Y 403.628,Z 836.352,A -85,B 0,C 180,E1 9975.425,E2 9975.425} C_VEL
LIN {X 0,Y 402.864,Z 847.126,A -85,B 0,C 180,E1 9980.298,E2 9980.298} C_VEL
LIN {X 0,Y 402.476,Z 853.882,A -85,B 0,C 180,E1 9985.701,E2 9985.701} C_VEL
LIN {X 0,Y 402.562,Z 855.611,A -85,B 0,C 180,E1 9990.002,E2 9990.002} C_VEL
LIN {X 0,Y 402.51,Z 853.016,A -85,B 0,C 180,E1 9995.38,E2 9995.38} C_VEL
LIN {X 0,Y 402.913,Z 845.197,A -85,B 0,C 180,E1 10000.795,E2 10000.795} C_VEL
LIN {X 0,Y 404.104,Z 831.765,A -85,B 0,C 180,E1 10006.266,E2 10006.266} C_VEL
LIN {X 0,Y 406.718,Z 811.943,A -85,B 0,C 180,E1 10011.78,E2 10011.78} C_VEL
LIN {X 0,Y 410.864,Z 787.351,A -85,B 0,C 180,E1 10016.74,E2 10016.74} C_VEL
LIN {X 0,Y 416.194,Z 757.512,A -85,B 0,C 180,E1 10021.202,E2 10021.202} C_VEL
LIN {X 0,Y 422.183,Z 724.216,A -85,B 0,C 180,E1 10024.884,E2 10024.884} C_VEL
LIN {X 0,Y 427.892,Z 688.644,A -85,B 0,C 180,E1 10027.743,E2 10027.743} C_VEL
LIN {X 0,Y 432.623,Z 652.241,A -85,B 0,C 180,E1 10029.786,E2 10029.786} C_VEL
LIN {X 0,Y 435.477,Z 618.018,A -85,B 0,C 180,E1 10031.079,E2 10031.079} C_VEL
LIN {X 0,Y 417.699,Z 580.356,A -85,B 0,C 180,E1 10034.032,E2 10034.032} C_VEL
LIN {X 0,Y 401.24,Z 550.852,A -85,B 0,C 180,E1 10036.76,E2 10036.76} C_VEL
LIN {X 0,Y 401.107,Z 549.53,A -85,B 0,C 180,E1 10036.95,E2 10036.95} C_VEL
LIN {X 0,Y 401.033,Z 549.53,A -85,B 0,C 180,E1 10042.971,E2 10042.971} C_VEL
LIN {X 0,Y 401.046,Z 549.53,A -85,B 0,C 180,E1 10049.934,E2 10049.934} C_VEL
LIN {X 0,Y 401.264,Z 549.53,A -85,B 0,C 180,E1 10055.551,E2 10055.551} C_VEL
LIN {X 0,Y 401.544,Z 549.53,A -85,B 0,C 180,E1 10062.489,E2 10062.489} C_VEL
LIN {X 0,Y 401.747,Z 549.53,A -85,B 0,C 180,E1 10069.16,E2 10069.16} C_VEL
LIN {X 0,Y 402.15,Z 549.53,A -85,B 0,C 180,E1 10075.679,E2 10075.679} C_VEL
LIN {X 0,Y 402.264,Z 549.53,A -85,B 0,C 180,E1 10082.131,E2 10082.131} C_VEL
LIN {X 0,Y 401.963,Z 549.53,A -85,B 0,C 180,E1 10088.616,E2 10088.616} C_VEL
LIN {X 0,Y 401.737,Z 549.53,A -85,B 0,C 180,E1 10095.222,E2 10095.222} C_VEL
LIN {X 0,Y 401.45,Z 549.53,A -85,B 0,C 180,E1 10102.055,E2 10102.055} C_VEL
LIN {X 0,Y 401.219,Z 549.53,A -85,B 0,C 180,E1 10109.243,E2 10109.243} C_VEL
LIN {X 0,Y 401.206,Z 549.53,A -85,B 0,C 180,E1 10114.314,E2 10114.314} C_VEL
LIN {X 0,Y 400.996,Z 549.53,A -85,B 0,C 180,E1 10121.179,E2 10121.179} C_VEL
LIN {X 0,Y 400.974,Z 549.53,A -85,B 0,C 180,E1 10127.357,E2 10127.357} C_VEL
LIN {X 0,Y 401.097,Z 549.53,A -85,B 0,C 180,E1 10132.988,E2 10132.988} C_VEL
LIN {X 0,Y 401.172,Z 549.53,A -85,B 0,C 180,E1 10139.841,E2 10139.841} C_VEL
LIN {X 0,Y 401.347,Z 549.53,A -85,B 0,C 180,E1 10145.568,E2 10145.568} C_VEL
LIN {X 0,Y 401.56,Z 549.53,A -85,B 0,C 180,E1 10152.503,E2 10152.503} C_VEL
LIN {X 0,Y 401.764,Z 550.317,A -85,B 0,C 180,E1 10155.42,E2 10155.42} C_VEL
LIN {X 0,Y 420.418,Z 587.678,A -85,B 0,C 180,E1 10158.82,E2 10158.82} C_VEL
LIN {X 0,Y 429.185,Z 610.909,A -85,B 0,C 180,E1 10160.927,E2 10160.927} C_VEL
LIN {X 0,Y 424.812,Z 646.125,A -85,B 0,C 180,E1 10163.036,E2 10163.036} C_VEL
LIN {X 0,Y 419.681,Z 678.52,A -85,B 0,C 180,E1 10165.875,E2 10165.875} C_VEL
LIN {X 0,Y 414.579,Z 707.23,A -85,B 0,C 180,E1 10169.364,E2 10169.364} C_VEL
LIN {X 0,Y 409.994,Z 731.813,A -85,B 0,C 180,E1 10173.427,E2 10173.427} C_VEL
LIN {X 0,Y 406.525,Z 751.976,A -85,B 0,C 180,E1 10178,E2 10178} C_VEL
LIN {X 0,Y 404.193,Z 767.297,A -85,B 0,C 180,E1 10182.943,E2 10182.943} C_VEL
LIN {X 0,Y 403.241,Z 776.463,A -85,B 0,C 180,E1 10187.419,E2 10187.419} C_VEL
LIN {X 0,Y 402.395,Z 781.828,A -85,B 0,C 180,E1 10192.023,E2 10192.023} C_VEL
LIN {X 0,Y 402.155,Z 783.266,A -85,B 0,C 180,E1 10196.76,E2 10196.76} C_VEL
LIN {X 0,Y 402.797,Z 780.445,A -85,B 0,C 180,E1 10201.632,E2 10201.632} C_VEL
LIN {X 0,Y 403.699,Z 772.77,A -85,B 0,C 180,E1 10206.73,E2 10206.73} C_VEL
LIN {X 0,Y 405.586,Z 759.151,A -85,B 0,C 180,E1 10212.042,E2 10212.042} C_VEL
LIN {X 0,Y 408.819,Z 740.465,A -85,B 0,C 180,E1 10216.925,E2 10216.925} C_VEL
LIN {X 0,Y 413.413,Z 716.365,A -85,B 0,C 180,E1 10221.402,E2 10221.402} C_VEL
LIN {X 0,Y 418.771,Z 688.338,A -85,B 0,C 180,E1 10225.181,E2 10225.181} C_VEL
LIN {X 0,Y 424.172,Z 656.678,A -85,B 0,C 180,E1 10228.264,E2 10228.264} C_VEL
LIN {X 0,Y 428.882,Z 622.501,A -85,B 0,C 180,E1 10230.586,E2 10230.586} C_VEL
LIN {X 0,Y 429.699,Z 611.506,A -85,B 0,C 180,E1 10231.202,E2 10231.202} C_VEL
LIN {X 0,Y 416.877,Z 579.373,A -85,B 0,C 180,E1 10234.28,E2 10234.28} C_VEL
LIN {X 0,Y 401.475,Z 550.255,A -85,B 0,C 180,E1 10237.238,E2 10237.238} C_VEL
LIN {X 0,Y 401.562,Z 549.53,A -85,B 0,C 180,E1 10242.528,E2 10242.528} C_VEL
LIN {X 0,Y 401.76,Z 549.53,A -85,B 0,C 180,E1 10249.196,E2 10249.196} C_VEL
LIN {X 0,Y 402.142,Z 549.53,A -85,B 0,C 180,E1 10255.715,E2 10255.715} C_VEL
LIN {X 0,Y 402.235,Z 549.53,A -85,B 0,C 180,E1 10262.167,E2 10262.167} C_VEL
LIN {X 0,Y 401.941,Z 549.53,A -85,B 0,C 180,E1 10268.653,E2 10268.653} C_VEL
LIN {X 0,Y 401.749,Z 549.53,A -85,B 0,C 180,E1 10275.259,E2 10275.259} C_VEL
LIN {X 0,Y 401.444,Z 549.53,A -85,B 0,C 180,E1 10282.094,E2 10282.094} C_VEL
LIN {X 0,Y 401.212,Z 549.53,A -85,B 0,C 180,E1 10289.284,E2 10289.284} C_VEL
LIN {X 0,Y 401.208,Z 549.53,A -85,B 0,C 180,E1 10294.358,E2 10294.358} C_VEL
LIN {X 0,Y 400.939,Z 549.53,A -85,B 0,C 180,E1 10301.174,E2 10301.174} C_VEL
LIN {X 0,Y 401.007,Z 549.819,A -85,B 0,C 180,E1 10303.001,E2 10303.001} C_VEL
LIN {X 0,Y 403.533,Z 555.305,A -85,B 0,C 180,E1 10303.502,E2 10303.502} C_VEL
LIN {X 0,Y 424.117,Z 592.297,A -85,B 0,C 180,E1 10307.006,E2 10307.006} C_VEL
LIN {X 0,Y 435.412,Z 619.792,A -85,B 0,C 180,E1 10309.072,E2 10309.072} C_VEL
LIN {X 0,Y 431.45,Z 659.309,A -85,B 0,C 180,E1 10310.622,E2 10310.622} C_VEL
